ABB RobotStudio station: stationlab5.rsstn

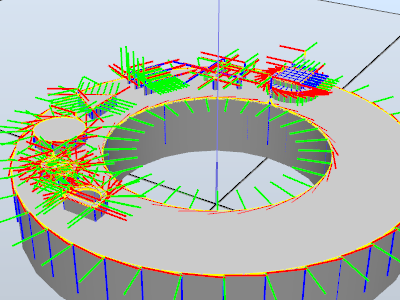
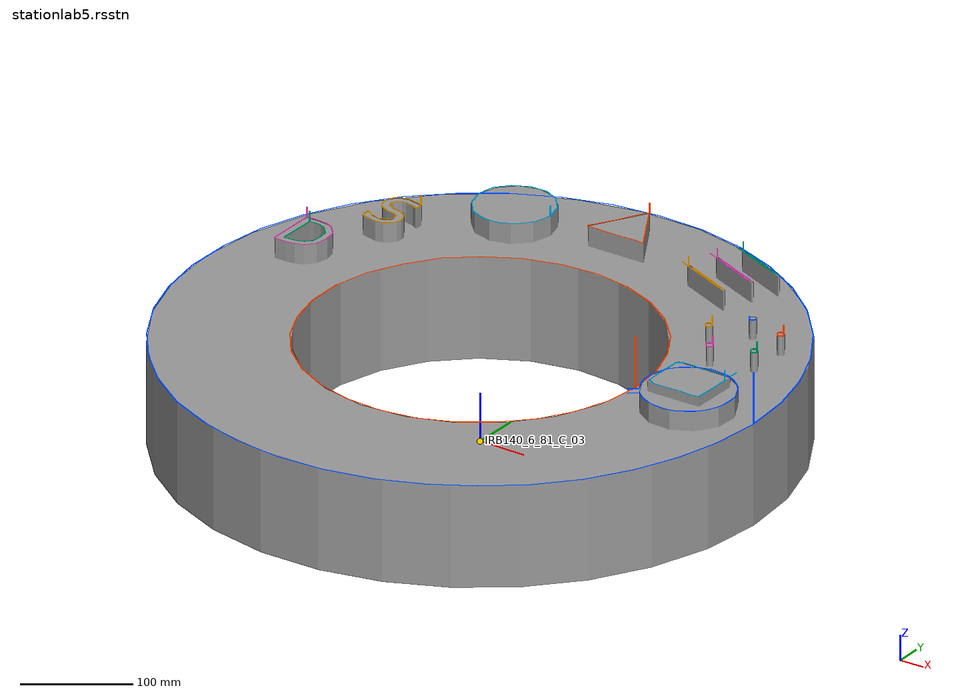
[picture v1: parts stored in the station drawn from their meshes, with robot base, taught points and paths (robot models come from the ABB library and are not in the file)]
Station Station (saved by RobotStudio 22.2.9947.0)
Controller lab5_controller
  mechanical unit ROB_1: IRB140_6_81_C_03, 6 joints, base frame (0, 0, 0) mm
Layout (positions relative to the parent item):
  - IRB140_6_81_C_03 [mechanism, from Robots\IRB140_6_81_C_G_03.rslib] at (0, 0, 0) mm; joint values [0, 0, 0, 0, 0.5236, 0] (rad or m)
  - ToolM_DS109 [mechanism, from Lab1\ToolM_DS109.rslib] at (506.29, 0, 679.5) mm, rotated rx 180 ry 60 rz 180 deg
  - lab5CADfiguras [part], size 590 x 586.8 x 130 mm
Attachment: ToolM_DS109 is attached to IRB140_6_81_C_03 / Link6
Attachment: Workobject_2 is attached to lab5CADfiguras
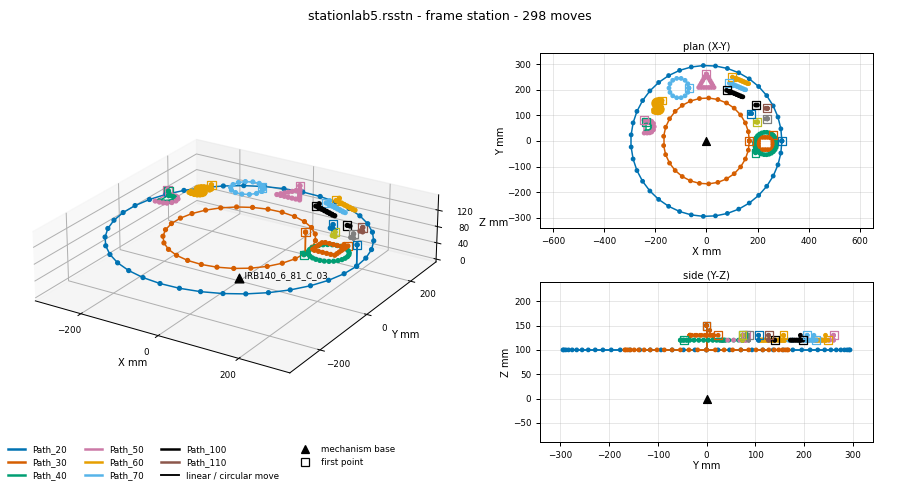
[picture p0: tool path of stationlab5.rsstn in frame station, 298 of 298 moves have a stored position in this frame; points joined in program order, loops and branches not executed]
Targets, tools, work objects and paths stored in the station, written as RAPID:
! task T_ROB1
MODULE CalibData
  PERS tooldata ToolM_DS109:=[TRUE,[[0,0,199.132],[0.949782708,0.067451832,-0.305553692,-0.000003594]],[0.13,[-0.003,72.016,0.062],[1,0,0,0],0,0,0]];
  TASK PERS wobjdata Workobject_1:=[FALSE,TRUE,"",[[0,0,0],[1,0,0,0]],[[0,0,0],[1,0,0,0]]];
  TASK PERS wobjdata Workobject_2:=[FALSE,TRUE,"",[[0,0,0],[1,0,0,0]],[[0,0,0],[1,0,0,0]]];
ENDMODULE

! task T_ROB1
MODULE Module1
  CONST robtarget Target_80_outter_ring_starts:=[[295,0,150],[0,0.707106781,0.707106781,0],[0,0,0,0],[9E+09,9E+09,9E+09,9E+09,9E+09,9E+09]];
  CONST robtarget Target_90:=[[295,0,100],[0,0.707106781,0.707106781,0],[0,0,0,0],[9E+09,9E+09,9E+09,9E+09,9E+09,9E+09]];
  CONST robtarget Target_100:=[[291.179827478,47.321327853,100],[0,0.647915395,0.761712308,0],[0,0,0,0],[9E+09,9E+09,9E+09,9E+09,9E+09,9E+09]];
  CONST robtarget Target_110:=[[279.818250374,93.417058171,100],[0,0.58452203,0.811377839,0],[0,0,0,0],[9E+09,9E+09,9E+09,9E+09,9E+09,9E+09]];
  CONST robtarget Target_120:=[[261.209527568,137.093335753,100],[0,0.517337814,0.855781272,0],[0,0,0,0],[9E+09,9E+09,9E+09,9E+09,9E+09,9E+09]];
  CONST robtarget Target_130:=[[235.835615204,177.21896795,100],[0,0.446798465,0.894634636,0],[0,0,0,0],[9E+09,9E+09,9E+09,9E+09,9E+09,9E+09]];
  CONST robtarget Target_140:=[[204.353684285,212.754721966,100],[0,0.373361455,0.927685951,0],[0,0,0,0],[9E+09,9E+09,9E+09,9E+09,9E+09,9E+09]];
  CONST robtarget Target_150:=[[167.579100286,242.780240439,100],[0,0.297503054,0.954720867,0],[0,0,0,0],[9E+09,9E+09,9E+09,9E+09,9E+09,9E+09]];
  CONST robtarget Target_160:=[[126.464305614,266.51787821,100],[0,0.219715231,0.975564051,0],[0,0,0,0],[9E+09,9E+09,9E+09,9E+09,9E+09,9E+09]];
  CONST robtarget Target_170:=[[82.074151855,283.352842931,100],[0,0.14050247,0.990080328,0],[0,0,0,0],[9E+09,9E+09,9E+09,9E+09,9E+09,9E+09]];
  CONST robtarget Target_180:=[[35.558320675,292.849117859,100],[0,0.060378497,0.998175554,0],[0,0,0,0],[9E+09,9E+09,9E+09,9E+09,9E+09,9E+09]];
  CONST robtarget Target_190:=[[-11.878452332,294.760754461,100],[0,-0.020137053,0.999797229,0],[0,0,0,0],[9E+09,9E+09,9E+09,9E+09,9E+09,9E+09]];
  CONST robtarget Target_200:=[[-59.007579664,289.038242352,100],[0,-0.100522007,0.994934835,0],[0,0,0,0],[9E+09,9E+09,9E+09,9E+09,9E+09,9E+09]];
  CONST robtarget Target_210:=[[-104.608441678,275.829791592,100],[0,-0.180255038,0.983619907,0],[0,0,0,0],[9E+09,9E+09,9E+09,9E+09,9E+09,9E+09]];
  CONST robtarget Target_220:=[[-147.5,255.477494116,100],[0,-0.258819045,0.965925826,0],[0,0,0,0],[9E+09,9E+09,9E+09,9E+09,9E+09,9E+09]];
  CONST robtarget Target_230:=[[-186.571385801,228.508463739,100],[0,-0.335704512,0.941967346,0],[0,0,0,0],[9E+09,9E+09,9E+09,9E+09,9E+09,9E+09]];
  CONST robtarget Target_240:=[[-220.81067071,195.621184181,100],[0,-0.410412805,0.911899846,0],[0,0,0,0],[9E+09,9E+09,9E+09,9E+09,9E+09,9E+09]];
  CONST robtarget Target_250:=[[-249.331075235,157.667418708,100],[0,-0.482459415,0.875918326,0],[0,0,0,0],[9E+09,9E+09,9E+09,9E+09,9E+09,9E+09]];
  CONST robtarget Target_260:=[[-271.393935879,115.630149909,100],[0,-0.55137709,0.834256139,0],[0,0,0,0],[9E+09,9E+09,9E+09,9E+09,9E+09,9E+09]];
  CONST robtarget Target_270:=[[-286.427836141,70.598120965,100],[0,-0.616718873,0.787183481,0],[0,0,0,0],[9E+09,9E+09,9E+09,9E+09,9E+09,9E+09]];
  CONST robtarget Target_280_outter_ring_half:=[[-294.0434059,23.737637771,100],[0,-0.678060997,0.735005636,0],[0,0,0,0],[9E+09,9E+09,9E+09,9E+09,9E+09,9E+09]];
  CONST robtarget Target_290:=[[-294.0434059,-23.737637771,100],[0,0.735005636,-0.678060997,0],[0,0,0,0],[9E+09,9E+09,9E+09,9E+09,9E+09,9E+09]];
  CONST robtarget Target_300:=[[-286.427836141,-70.598120965,100],[0,0.787183481,-0.616718873,0],[0,0,0,0],[9E+09,9E+09,9E+09,9E+09,9E+09,9E+09]];
  CONST robtarget Target_310:=[[-271.393935879,-115.630149909,100],[0,0.834256139,-0.55137709,0],[0,0,0,0],[9E+09,9E+09,9E+09,9E+09,9E+09,9E+09]];
  CONST robtarget Target_320:=[[-249.331075235,-157.667418708,100],[0,0.875918326,-0.482459415,0],[0,0,0,0],[9E+09,9E+09,9E+09,9E+09,9E+09,9E+09]];
  CONST robtarget Target_330:=[[-220.81067071,-195.621184181,100],[0,0.911899846,-0.410412805,0],[0,0,0,0],[9E+09,9E+09,9E+09,9E+09,9E+09,9E+09]];
  CONST robtarget Target_340:=[[-186.571385801,-228.508463739,100],[0,0.941967346,-0.335704512,0],[0,0,0,0],[9E+09,9E+09,9E+09,9E+09,9E+09,9E+09]];
  CONST robtarget Target_350:=[[-147.5,-255.477494116,100],[0,0.965925826,-0.258819045,0],[0,0,0,0],[9E+09,9E+09,9E+09,9E+09,9E+09,9E+09]];
  CONST robtarget Target_360:=[[-104.608441678,-275.829791592,100],[0,0.983619907,-0.180255038,0],[0,0,0,0],[9E+09,9E+09,9E+09,9E+09,9E+09,9E+09]];
  CONST robtarget Target_370:=[[-59.007579664,-289.038242352,100],[0,0.994934835,-0.100522007,0],[0,0,0,0],[9E+09,9E+09,9E+09,9E+09,9E+09,9E+09]];
  CONST robtarget Target_380:=[[-11.878452332,-294.760754461,100],[0,0.999797229,-0.020137053,0],[0,0,0,0],[9E+09,9E+09,9E+09,9E+09,9E+09,9E+09]];
  CONST robtarget Target_390:=[[35.558320675,-292.849117859,100],[0,0.998175554,0.060378497,0],[0,0,0,0],[9E+09,9E+09,9E+09,9E+09,9E+09,9E+09]];
  CONST robtarget Target_400:=[[82.074151855,-283.352842931,100],[0,0.990080328,0.14050247,0],[0,0,0,0],[9E+09,9E+09,9E+09,9E+09,9E+09,9E+09]];
  CONST robtarget Target_410:=[[126.464305614,-266.51787821,100],[0,0.975564051,0.219715231,0],[0,0,0,0],[9E+09,9E+09,9E+09,9E+09,9E+09,9E+09]];
  CONST robtarget Target_420:=[[167.579100286,-242.780240439,100],[0,0.954720867,0.297503054,0],[0,0,0,0],[9E+09,9E+09,9E+09,9E+09,9E+09,9E+09]];
  CONST robtarget Target_430:=[[204.353684285,-212.754721966,100],[0,0.927685951,0.373361455,0],[0,0,0,0],[9E+09,9E+09,9E+09,9E+09,9E+09,9E+09]];
  CONST robtarget Target_440:=[[235.835615204,-177.21896795,100],[0,0.894634636,0.446798465,0],[0,0,0,0],[9E+09,9E+09,9E+09,9E+09,9E+09,9E+09]];
  CONST robtarget Target_450:=[[261.209527568,-137.093335753,100],[0,0.855781272,0.517337814,0],[0,0,0,0],[9E+09,9E+09,9E+09,9E+09,9E+09,9E+09]];
  CONST robtarget Target_460:=[[279.818250374,-93.417058171,100],[0,0.811377839,0.58452203,0],[0,0,0,0],[9E+09,9E+09,9E+09,9E+09,9E+09,9E+09]];
  CONST robtarget Target_470:=[[291.179827478,-47.321327853,100],[0,0.761712308,0.647915395,0],[0,0,0,0],[9E+09,9E+09,9E+09,9E+09,9E+09,9E+09]];
  CONST robtarget Target_480:=[[295,0,100],[0,0.707106781,0.707106781,0],[0,0,0,0],[9E+09,9E+09,9E+09,9E+09,9E+09,9E+09]];
  CONST robtarget Target_490_outer_ring_ends:=[[295,0,150],[0,0.707106781,0.707106781,0],[0,0,0,0],[9E+09,9E+09,9E+09,9E+09,9E+09,9E+09]];
  CONST robtarget Target_500_inner_ring_starts:=[[168,0,150],[0,-0.707106781,0.707106781,0],[0,0,0,0],[9E+09,9E+09,9E+09,9E+09,9E+09,9E+09]];
  CONST robtarget Target_510:=[[168,0,100],[0,-0.707106781,0.707106781,0],[0,0,0,0],[9E+09,9E+09,9E+09,9E+09,9E+09,9E+09]];
  CONST robtarget Target_520:=[[164.072253359,-36.115033955,100],[0,-0.62651,0.779413382,0],[0,0,0,0],[9E+09,9E+09,9E+09,9E+09,9E+09,9E+09]];
  CONST robtarget Target_530:=[[152.472670505,-70.541369062,100],[0,-0.538567962,0.842582074,0],[0,0,0,0],[9E+09,9E+09,9E+09,9E+09,9E+09,9E+09]];
  CONST robtarget Target_540:=[[133.743635039,-101.669268153,100],[0,-0.444311706,0.895872261,0],[0,0,0,0],[9E+09,9E+09,9E+09,9E+09,9E+09,9E+09]];
  CONST robtarget Target_550:=[[108.760895843,-128.043225261,100],[0,-0.344846303,0.938659165,0],[0,0,0,0],[9E+09,9E+09,9E+09,9E+09,9E+09,9E+09]];
  CONST robtarget Target_560:=[[78.692618038,-148.430023467,100],[0,-0.241337891,0.970441148,0],[0,0,0,0],[9E+09,9E+09,9E+09,9E+09,9E+09,9E+09]];
  CONST robtarget Target_570:=[[44.944760873,-161.876398743,100],[0,-0.135000014,0.990845597,0],[0,0,0,0],[9E+09,9E+09,9E+09,9E+09,9E+09,9E+09]];
  CONST robtarget Target_580:=[[9.095336642,-167.753613527,100],[0,-0.027079385,0.999633286,0],[0,0,0,0],[9E+09,9E+09,9E+09,9E+09,9E+09,9E+09]];
  CONST robtarget Target_590:=[[-27.179375421,-165.786855787,100],[0,0.081158726,0.99670119,0],[0,0,0,0],[9E+09,9E+09,9E+09,9E+09,9E+09,9E+09]];
  CONST robtarget Target_600:=[[-62.183210097,-156.068088929,100],[0,0.188445324,0.982083683,0],[0,0,0,0],[9E+09,9E+09,9E+09,9E+09,9E+09,9E+09]];
  CONST robtarget Target_610:=[[-94.279426981,-139.05175169,100],[0,0.293522573,0.955952143,0],[0,0,0,0],[9E+09,9E+09,9E+09,9E+09,9E+09,9E+09]];
  CONST robtarget Target_620:=[[-121.967242643,-115.533509087,100],[0,0.395158539,0.918612938,0],[0,0,0,0],[9E+09,9E+09,9E+09,9E+09,9E+09,9E+09]];
  CONST robtarget Target_630:=[[-143.952005596,-86.613048006,100],[0,0.492161631,0.870503836,0],[0,0,0,0],[9E+09,9E+09,9E+09,9E+09,9E+09,9E+09]];
  CONST robtarget Target_640:=[[-159.205732759,-53.642657063,100],[0,0.583394579,0.812188873,0],[0,0,0,0],[9E+09,9E+09,9E+09,9E+09,9E+09,9E+09]];
  CONST robtarget Target_650_inner_ring_half:=[[-167.015176802,-18.163995095,100],[0,0.667787759,0.744351738,0],[0,0,0,0],[9E+09,9E+09,9E+09,9E+09,9E+09,9E+09]];
  CONST robtarget Target_660:=[[-167.015176802,18.163995095,100],[0,0.744351738,0.667787759,0],[0,0,0,0],[9E+09,9E+09,9E+09,9E+09,9E+09,9E+09]];
  CONST robtarget Target_670:=[[-159.205732759,53.642657063,100],[0,0.812188873,0.583394579,0],[0,0,0,0],[9E+09,9E+09,9E+09,9E+09,9E+09,9E+09]];
  CONST robtarget Target_680:=[[-143.952005596,86.613048006,100],[0,0.870503836,0.492161631,0],[0,0,0,0],[9E+09,9E+09,9E+09,9E+09,9E+09,9E+09]];
  CONST robtarget Target_690:=[[-121.967242643,115.533509087,100],[0,0.918612938,0.395158539,0],[0,0,0,0],[9E+09,9E+09,9E+09,9E+09,9E+09,9E+09]];
  CONST robtarget Target_700:=[[-94.279426981,139.05175169,100],[0,0.955952143,0.293522573,0],[0,0,0,0],[9E+09,9E+09,9E+09,9E+09,9E+09,9E+09]];
  CONST robtarget Target_710:=[[-62.183210097,156.068088929,100],[0,0.982083683,0.188445324,0],[0,0,0,0],[9E+09,9E+09,9E+09,9E+09,9E+09,9E+09]];
  CONST robtarget Target_720:=[[-27.179375421,165.786855787,100],[0,0.99670119,0.081158726,0],[0,0,0,0],[9E+09,9E+09,9E+09,9E+09,9E+09,9E+09]];
  CONST robtarget Target_730:=[[9.095336642,167.753613527,100],[0,0.999633286,-0.027079385,0],[0,0,0,0],[9E+09,9E+09,9E+09,9E+09,9E+09,9E+09]];
  CONST robtarget Target_740:=[[44.944760873,161.876398743,100],[0,0.990845597,-0.135000014,0],[0,0,0,0],[9E+09,9E+09,9E+09,9E+09,9E+09,9E+09]];
  CONST robtarget Target_750:=[[78.692618038,148.430023467,100],[0,0.970441148,-0.241337891,0],[0,0,0,0],[9E+09,9E+09,9E+09,9E+09,9E+09,9E+09]];
  CONST robtarget Target_760:=[[108.760895843,128.043225261,100],[0,0.938659165,-0.344846303,0],[0,0,0,0],[9E+09,9E+09,9E+09,9E+09,9E+09,9E+09]];
  CONST robtarget Target_770:=[[133.743635039,101.669268153,100],[0,0.895872261,-0.444311706,0],[0,0,0,0],[9E+09,9E+09,9E+09,9E+09,9E+09,9E+09]];
  CONST robtarget Target_780:=[[152.472670505,70.541369062,100],[0,0.842582074,-0.538567962,0],[0,0,0,0],[9E+09,9E+09,9E+09,9E+09,9E+09,9E+09]];
  CONST robtarget Target_790:=[[164.072253359,36.115033955,100],[0,0.779413382,-0.62651,0],[0,0,0,0],[9E+09,9E+09,9E+09,9E+09,9E+09,9E+09]];
  CONST robtarget Target_800:=[[168,0,100],[0,-0.707106781,0.707106781,0],[0,0,0,0],[9E+09,9E+09,9E+09,9E+09,9E+09,9E+09]];
  CONST robtarget Target_810_inner_ring_ends:=[[168,0,150],[0,-0.707106781,0.707106781,0],[0,0,0,0],[9E+09,9E+09,9E+09,9E+09,9E+09,9E+09]];
  CONST robtarget Target_810:=[[-236.504880452,74.974751988,130],[0,-0.707106781,0.707106781,0],[0,0,0,0],[9E+09,9E+09,9E+09,9E+09,9E+09,9E+09]];
  CONST robtarget Target_820_d_inner_starts:=[[-236.504880452,74.974751988,120],[0,-0.707106781,0.707106781,0],[0,0,0,0],[9E+09,9E+09,9E+09,9E+09,9E+09,9E+09]];
  CONST robtarget Target_830:=[[-236.504880452,36.482045343,120],[0,-0.707106781,0.707106781,0],[0,0,0,0],[9E+09,9E+09,9E+09,9E+09,9E+09,9E+09]];
  CONST robtarget Target_840:=[[-231.440050631,36.482045343,120],[0,1,0,0],[0,0,0,0],[9E+09,9E+09,9E+09,9E+09,9E+09,9E+09]];
  CONST robtarget Target_850:=[[-223.680731344,37.191121518,120],[0,0.994543645,0.104321318,0],[0,0,0,0],[9E+09,9E+09,9E+09,9E+09,9E+09,9E+09]];
  CONST robtarget Target_860:=[[-217.623194877,39.804573706,120],[0,0.953587299,0.301116693,0],[0,0,0,0],[9E+09,9E+09,9E+09,9E+09,9E+09,9E+09]];
  CONST robtarget Target_870:=[[-212.396290501,46.044444047,120],[0,0.839280324,0.54369894,0],[0,0,0,0],[9E+09,9E+09,9E+09,9E+09,9E+09,9E+09]];
  CONST robtarget Target_880:=[[-210.653989042,55.768917304,120],[0,0.707106781,0.707106781,0],[0,0,0,0],[9E+09,9E+09,9E+09,9E+09,9E+09,9E+09]];
  CONST robtarget Target_890:=[[-212.558365055,65.594687159,120],[0,0.536830761,0.843689951,0],[0,0,0,0],[9E+09,9E+09,9E+09,9E+09,9E+09,9E+09]];
  CONST robtarget Target_900:=[[-218.230974456,71.976372734,120],[0,0.271476286,0.962445129,0],[0,0,0,0],[9E+09,9E+09,9E+09,9E+09,9E+09,9E+09]];
  CONST robtarget Target_910:=[[-223.923843175,74.265675813,120],[0,0.115102592,0.993353609,0],[0,0,0,0],[9E+09,9E+09,9E+09,9E+09,9E+09,9E+09]];
  CONST robtarget Target_920:=[[-231.440050631,74.974751988,120],[0,0,1,0],[0,0,0,0],[9E+09,9E+09,9E+09,9E+09,9E+09,9E+09]];
  CONST robtarget Target_930:=[[-236.504880452,74.974751988,120],[0,0,1,0],[0,0,0,0],[9E+09,9E+09,9E+09,9E+09,9E+09,9E+09]];
  CONST robtarget Target_940_d_inner:=[[-236.504880452,74.974751988,130],[0,0,1,0],[0,0,0,0],[9E+09,9E+09,9E+09,9E+09,9E+09,9E+09]];
  CONST robtarget Target_940:=[[-243.149937179,80.728398666,130],[0,-0.707106781,0.707106781,0],[0,0,0,0],[9E+09,9E+09,9E+09,9E+09,9E+09,9E+09]];
  CONST robtarget Target_950_d_outter_starts:=[[-243.149937179,80.728398666,120],[0,-0.707106781,0.707106781,0],[0,0,0,0],[9E+09,9E+09,9E+09,9E+09,9E+09,9E+09]];
  CONST robtarget Target_960:=[[-243.149937179,30.728398666,120],[0,-0.707106781,0.707106781,0],[0,0,0,0],[9E+09,9E+09,9E+09,9E+09,9E+09,9E+09]];
  CONST robtarget Target_970:=[[-231.642643824,30.728398666,120],[0,1,0,0],[0,0,0,0],[9E+09,9E+09,9E+09,9E+09,9E+09,9E+09]];
  CONST robtarget Target_980:=[[-221.654799415,31.538771437,120],[0,0.994784133,0.102002596,0],[0,0,0,0],[9E+09,9E+09,9E+09,9E+09,9E+09,9E+09]];
  CONST robtarget Target_990:=[[-213.935998767,34.739743885,120],[0,0.960985001,0.276600484,0],[0,0,0,0],[9E+09,9E+09,9E+09,9E+09,9E+09,9E+09]];
  CONST robtarget Target_1000:=[[-206.500828589,43.329695262,120],[0,0.851421887,0.524481429,0],[0,0,0,0],[9E+09,9E+09,9E+09,9E+09,9E+09,9E+09]];
  CONST robtarget Target_1010:=[[-203.725301846,55.687880027,120],[0,0.707106781,0.707106781,0],[0,0,0,0],[9E+09,9E+09,9E+09,9E+09,9E+09,9E+09]];
  CONST robtarget Target_1020:=[[-206.379272673,68.268917304,120],[0,0.525079618,0.851053109,0],[0,0,0,0],[9E+09,9E+09,9E+09,9E+09,9E+09,9E+09]];
  CONST robtarget Target_1030:=[[-213.85496149,76.757572086,120],[0,0.288854798,0.957372919,0],[0,0,0,0],[9E+09,9E+09,9E+09,9E+09,9E+09,9E+09]];
  CONST robtarget Target_1040:=[[-220.702611409,79.674914063,120],[0,0.128060594,0.991766346,0],[0,0,0,0],[9E+09,9E+09,9E+09,9E+09,9E+09,9E+09]];
  CONST robtarget Target_1050:=[[-231.764199739,80.728398666,120],[0,0,1,0],[0,0,0,0],[9E+09,9E+09,9E+09,9E+09,9E+09,9E+09]];
  CONST robtarget Target_1060:=[[-243.149937179,80.728398666,120],[0,0,1,0],[0,0,0,0],[9E+09,9E+09,9E+09,9E+09,9E+09,9E+09]];
  CONST robtarget Target_1070_d_outter_ends:=[[-243.149937179,80.728398666,130],[0,0,1,0],[0,0,0,0],[9E+09,9E+09,9E+09,9E+09,9E+09,9E+09]];
  CONST robtarget Target_1070:=[[-174.142803292,158.219300938,130],[0,0.227282029,0.973828978,0],[0,0,0,0],[9E+09,9E+09,9E+09,9E+09,9E+09,9E+09]];
  CONST robtarget Target_1080_s_starts:=[[-174.142803292,158.219300938,120],[0,0.227282029,0.973828978,0],[0,0,0,0],[9E+09,9E+09,9E+09,9E+09,9E+09,9E+09]];
  CONST robtarget Target_1090:=[[-181.071490488,160.630159933,120],[0,0.109402737,0.993997506,0],[0,0,0,0],[9E+09,9E+09,9E+09,9E+09,9E+09,9E+09]];
  CONST robtarget Target_1100:=[[-189.013143649,161.460792024,120],[0,0,1,0],[0,0,0,0],[9E+09,9E+09,9E+09,9E+09,9E+09,9E+09]];
  CONST robtarget Target_1110:=[[-195.698719013,160.43263157,120],[0,-0.163403874,0.98655926,0],[0,0,0,0],[9E+09,9E+09,9E+09,9E+09,9E+09,9E+09]];
  CONST robtarget Target_1120:=[[-201.087697944,157.348150208,120],[0,-0.349735999,0.936848297,0],[0,0,0,0],[9E+09,9E+09,9E+09,9E+09,9E+09,9E+09]];
  CONST robtarget Target_1130:=[[-204.643208478,152.7442199,120],[0,-0.537680352,0.843148764,0],[0,0,0,0],[9E+09,9E+09,9E+09,9E+09,9E+09,9E+09]];
  CONST robtarget Target_1140:=[[-205.828378657,147.157712607,120],[0,-0.707106781,0.707106781,0],[0,0,0,0],[9E+09,9E+09,9E+09,9E+09,9E+09,9E+09]];
  CONST robtarget Target_1150:=[[-204.977487247,142.011845508,120],[0,0.823620533,-0.567141267,0],[0,0,0,0],[9E+09,9E+09,9E+09,9E+09,9E+09,9E+09]];
  CONST robtarget Target_1160:=[[-202.586887571,138.122056205,120],[0,0.916450944,-0.400147057,0],[0,0,0,0],[9E+09,9E+09,9E+09,9E+09,9E+09,9E+09]];
  CONST robtarget Target_1170:=[[-198.960469418,135.42756674,120],[0,0.972793034,-0.231675878,0],[0,0,0,0],[9E+09,9E+09,9E+09,9E+09,9E+09,9E+09]];
  CONST robtarget Target_1180:=[[-194.321085302,133.705524601,120],[0,0.991585883,-0.129450518,0],[0,0,0,0],[9E+09,9E+09,9E+09,9E+09,9E+09,9E+09]];
  CONST robtarget Target_1190:=[[-185.2854289,131.43648084,120],[0,0.990653418,-0.136403098,0],[0,0,0,0],[9E+09,9E+09,9E+09,9E+09,9E+09,9E+09]];
  CONST robtarget Target_1200:=[[-180.605526145,128.640694779,120],[0,0.900437375,-0.43498567,0],[0,0,0,0],[9E+09,9E+09,9E+09,9E+09,9E+09,9E+09]];
  CONST robtarget Target_1210:=[[-179.126595837,123.77845815,120],[0,-0.707106781,0.707106781,0],[0,0,0,0],[9E+09,9E+09,9E+09,9E+09,9E+09,9E+09]];
  CONST robtarget Target_1220:=[[-181.942641218,117.720921683,120],[0,-0.334706425,0.942322455,0],[0,0,0,0],[9E+09,9E+09,9E+09,9E+09,9E+09,9E+09]];
  CONST robtarget Target_1230:=[[-190.269221444,115.431618604,120],[0,0,1,0],[0,0,0,0],[9E+09,9E+09,9E+09,9E+09,9E+09,9E+09]];
  CONST robtarget Target_1240:=[[-198.271652563,117.133401424,120],[0,0.193221244,0.981155212,0],[0,0,0,0],[9E+09,9E+09,9E+09,9E+09,9E+09,9E+09]];
  CONST robtarget Target_1250:=[[-205.706822741,121.914600776,120],[0,0.367929084,0.929853854,0],[0,0,0,0],[9E+09,9E+09,9E+09,9E+09,9E+09,9E+09]];
  CONST robtarget Target_1260:=[[-206.193046404,121.914600776,120],[0,0,1,0],[0,0,0,0],[9E+09,9E+09,9E+09,9E+09,9E+09,9E+09]];
  CONST robtarget Target_1270:=[[-206.193046404,113.567761229,120],[0,-0.707106781,0.707106781,0],[0,0,0,0],[9E+09,9E+09,9E+09,9E+09,9E+09,9E+09]];
  CONST robtarget Target_1280:=[[-199.021247376,110.812493806,120],[0,0.989541733,-0.144246866,0],[0,0,0,0],[9E+09,9E+09,9E+09,9E+09,9E+09,9E+09]];
  CONST robtarget Target_1290:=[[-189.782997782,109.677971926,120],[0,1,0,0],[0,0,0,0],[9E+09,9E+09,9E+09,9E+09,9E+09,9E+09]];
  CONST robtarget Target_1300:=[[-182.16549373,110.853012445,120],[0,0.983031812,0.183435159,0],[0,0,0,0],[9E+09,9E+09,9E+09,9E+09,9E+09,9E+09]];
  CONST robtarget Target_1310:=[[-176.735996161,114.216059447,120],[0,0.932113972,0.362165078,0],[0,0,0,0],[9E+09,9E+09,9E+09,9E+09,9E+09,9E+09]];
  CONST robtarget Target_1320:=[[-173.393208478,119.037777437,120],[0,0.833172024,0.553013904,0],[0,0,0,0],[9E+09,9E+09,9E+09,9E+09,9E+09,9E+09]];
  CONST robtarget Target_1330:=[[-172.197908641,124.831942753,120],[0,0.707106781,0.707106781,0],[0,0,0,0],[9E+09,9E+09,9E+09,9E+09,9E+09,9E+09]];
  CONST robtarget Target_1340:=[[-174.588508316,132.672299317,120],[0,0.446758127,0.89465478,0],[0,0,0,0],[9E+09,9E+09,9E+09,9E+09,9E+09,9E+09]];
  CONST robtarget Target_1350:=[[-182.124975091,137.433239349,120],[0,0.148422353,0.988924064,0],[0,0,0,0],[9E+09,9E+09,9E+09,9E+09,9E+09,9E+09]];
  CONST robtarget Target_1360:=[[-192.37619065,140.066950857,120],[0,0.131118728,0.991366672,0],[0,0,0,0],[9E+09,9E+09,9E+09,9E+09,9E+09,9E+09]];
  CONST robtarget Target_1370:=[[-197.21816796,142.80195896,120],[0,0.408744216,0.912648983,0],[0,0,0,0],[9E+09,9E+09,9E+09,9E+09,9E+09,9E+09]];
  CONST robtarget Target_1380:=[[-198.899691461,147.846529463,120],[0,0.707106781,0.707106781,0],[0,0,0,0],[9E+09,9E+09,9E+09,9E+09,9E+09,9E+09]];
  CONST robtarget Target_1390:=[[-196.043127441,153.539398182,120],[0,0.947786225,0.318906369,0],[0,0,0,0],[9E+09,9E+09,9E+09,9E+09,9E+09,9E+09]];
  CONST robtarget Target_1400:=[[-188.567438624,155.707145346,120],[0,1,0,0],[0,0,0,0],[9E+09,9E+09,9E+09,9E+09,9E+09,9E+09]];
  CONST robtarget Target_1410:=[[-180.74734138,154.086399803,120],[0,0.979048021,-0.203629497,0],[0,0,0,0],[9E+09,9E+09,9E+09,9E+09,9E+09,9E+09]];
  CONST robtarget Target_1420:=[[-174.142803292,150.277647777,120],[0,1,0,0],[0,0,0,0],[9E+09,9E+09,9E+09,9E+09,9E+09,9E+09]];
  CONST robtarget Target_1430:=[[-174.142803292,158.219300938,120],[0,0.707106781,0.707106781,0],[0,0,0,0],[9E+09,9E+09,9E+09,9E+09,9E+09,9E+09]];
  CONST robtarget Target_1440_s_ends:=[[-174.142803292,158.219300938,130],[0,0.707106781,0.707106781,0],[0,0,0,0],[9E+09,9E+09,9E+09,9E+09,9E+09,9E+09]];
  CONST robtarget Target_1440:=[[-68.753776769,206.725037499,130],[0,0.707106781,0.707106781,0],[0,0,0,0],[9E+09,9E+09,9E+09,9E+09,9E+09,9E+09]];
  CONST robtarget Target_1450_circle_starts:=[[-68.753776769,206.725037499,120],[0,0.707106781,0.707106781,0],[0,0,0,0],[9E+09,9E+09,9E+09,9E+09,9E+09,9E+09]];
  CONST robtarget Target_1460:=[[-72.586344164,223.516612395,120],[0,0.532032077,0.846724199,0],[0,0,0,0],[9E+09,9E+09,9E+09,9E+09,9E+09,9E+09]];
  CONST robtarget Target_1470:=[[-83.324959372,236.982409948,120],[0,0.330279062,0.94388333,0],[0,0,0,0],[9E+09,9E+09,9E+09,9E+09,9E+09,9E+09]];
  CONST robtarget Target_1480:=[[-98.842707952,244.455363805,120],[0,0.111964476,0.99371221,0],[0,0,0,0],[9E+09,9E+09,9E+09,9E+09,9E+09,9E+09]];
  CONST robtarget Target_1490:=[[-116.066109483,244.455363805,120],[0,-0.111964476,0.99371221,0],[0,0,0,0],[9E+09,9E+09,9E+09,9E+09,9E+09,9E+09]];
  CONST robtarget Target_1500:=[[-131.583858063,236.982409948,120],[0,-0.330279062,0.94388333,0],[0,0,0,0],[9E+09,9E+09,9E+09,9E+09,9E+09,9E+09]];
  CONST robtarget Target_1510:=[[-142.322473271,223.516612395,120],[0,-0.532032077,0.846724199,0],[0,0,0,0],[9E+09,9E+09,9E+09,9E+09,9E+09,9E+09]];
  CONST robtarget Target_1520:=[[-146.155040666,206.725037499,120],[0,-0.707106781,0.707106781,0],[0,0,0,0],[9E+09,9E+09,9E+09,9E+09,9E+09,9E+09]];
  CONST robtarget Target_1530:=[[-142.322473271,189.933462603,120],[0,0.846724199,-0.532032077,0],[0,0,0,0],[9E+09,9E+09,9E+09,9E+09,9E+09,9E+09]];
  CONST robtarget Target_1540:=[[-131.583858063,176.46766505,120],[0,0.94388333,-0.330279062,0],[0,0,0,0],[9E+09,9E+09,9E+09,9E+09,9E+09,9E+09]];
  CONST robtarget Target_1550:=[[-116.066109483,168.994711193,120],[0,0.99371221,-0.111964476,0],[0,0,0,0],[9E+09,9E+09,9E+09,9E+09,9E+09,9E+09]];
  CONST robtarget Target_1560:=[[-98.842707952,168.994711193,120],[0,0.99371221,0.111964476,0],[0,0,0,0],[9E+09,9E+09,9E+09,9E+09,9E+09,9E+09]];
  CONST robtarget Target_1570:=[[-83.324959372,176.46766505,120],[0,0.94388333,0.330279062,0],[0,0,0,0],[9E+09,9E+09,9E+09,9E+09,9E+09,9E+09]];
  CONST robtarget Target_1580:=[[-72.586344164,189.933462603,120],[0,0.846724199,0.532032077,0],[0,0,0,0],[9E+09,9E+09,9E+09,9E+09,9E+09,9E+09]];
  CONST robtarget Target_1590:=[[-68.753776769,206.725037499,120],[0,0.707106781,0.707106781,0],[0,0,0,0],[9E+09,9E+09,9E+09,9E+09,9E+09,9E+09]];
  CONST robtarget Target_1600_circle_ends:=[[-68.753776769,206.725037499,130],[0,0.707106781,0.707106781,0],[0,0,0,0],[9E+09,9E+09,9E+09,9E+09,9E+09,9E+09]];
  CONST robtarget Target_2450_point1_starts:=[[195.937959768,143.518538082,120],[0,0,-0.707106781,0.707106781],[0,0,0,0],[9E+09,9E+09,9E+09,9E+09,9E+09,9E+09]];
  CONST robtarget Target_2460:=[[192.506872882,140.087451197,120],[0.5,-0.5,0.5,-0.5],[0,0,0,0],[9E+09,9E+09,9E+09,9E+09,9E+09,9E+09]];
  CONST robtarget Target_2470:=[[195.937959768,136.656364312,120],[0.707106781,-0.707106781,0,0],[0,0,0,0],[9E+09,9E+09,9E+09,9E+09,9E+09,9E+09]];
  CONST robtarget Target_2480_point1_ends:=[[199.369046653,140.087451197,120],[0.5,-0.5,-0.5,0.5],[0,0,0,0],[9E+09,9E+09,9E+09,9E+09,9E+09,9E+09]];
  CONST robtarget Target_2480:=[[238.2927152,127.440384636,130],[0,0.707106781,0.707106781,0],[0,0,0,0],[9E+09,9E+09,9E+09,9E+09,9E+09,9E+09]];
  CONST robtarget Target_2490_point2_starts:=[[238.2927152,127.440384636,120],[0,0.707106781,0.707106781,0],[0,0,0,0],[9E+09,9E+09,9E+09,9E+09,9E+09,9E+09]];
  CONST robtarget Target_2500:=[[234.861628315,130.871471522,120],[0,0,1,0],[0,0,0,0],[9E+09,9E+09,9E+09,9E+09,9E+09,9E+09]];
  CONST robtarget Target_2510:=[[231.430541429,127.440384636,120],[0,-0.707106781,0.707106781,0],[0,0,0,0],[9E+09,9E+09,9E+09,9E+09,9E+09,9E+09]];
  CONST robtarget Target_2520:=[[234.861628315,124.009297751,120],[0,1,0,0],[0,0,0,0],[9E+09,9E+09,9E+09,9E+09,9E+09,9E+09]];
  CONST robtarget Target_2530:=[[238.2927152,127.440384636,120],[0,0.707106781,0.707106781,0],[0,0,0,0],[9E+09,9E+09,9E+09,9E+09,9E+09,9E+09]];
  CONST robtarget Target_2540_point2_ends:=[[238.2927152,127.440384636,130],[0,0.707106781,0.707106781,0],[0,0,0,0],[9E+09,9E+09,9E+09,9E+09,9E+09,9E+09]];
  CONST robtarget Target_2540:=[[238.2927152,86.51361753,130],[0,0.707106781,0.707106781,0],[0,0,0,0],[9E+09,9E+09,9E+09,9E+09,9E+09,9E+09]];
  CONST robtarget Target_2550_point3_starts:=[[238.2927152,86.51361753,120],[0,0.707106781,0.707106781,0],[0,0,0,0],[9E+09,9E+09,9E+09,9E+09,9E+09,9E+09]];
  CONST robtarget Target_2560:=[[234.861628315,89.944704415,120],[0,0,1,0],[0,0,0,0],[9E+09,9E+09,9E+09,9E+09,9E+09,9E+09]];
  CONST robtarget Target_2570:=[[231.430541429,86.51361753,120],[0,-0.707106781,0.707106781,0],[0,0,0,0],[9E+09,9E+09,9E+09,9E+09,9E+09,9E+09]];
  CONST robtarget Target_2580:=[[234.861628315,83.082530645,120],[0,1,0,0],[0,0,0,0],[9E+09,9E+09,9E+09,9E+09,9E+09,9E+09]];
  CONST robtarget Target_2590:=[[238.2927152,86.51361753,120],[0,0.707106781,0.707106781,0],[0,0,0,0],[9E+09,9E+09,9E+09,9E+09,9E+09,9E+09]];
  CONST robtarget Target_2600_point3_ends:=[[238.2927152,86.51361753,130],[0,0.707106781,0.707106781,0],[0,0,0,0],[9E+09,9E+09,9E+09,9E+09,9E+09,9E+09]];
  CONST robtarget Target_2600:=[[199.369046653,73.86655097,130],[0,0.707106781,0.707106781,0],[0,0,0,0],[9E+09,9E+09,9E+09,9E+09,9E+09,9E+09]];
  CONST robtarget Target_2610_point4_starts:=[[199.369046653,73.86655097,120],[0,0.707106781,0.707106781,0],[0,0,0,0],[9E+09,9E+09,9E+09,9E+09,9E+09,9E+09]];
  CONST robtarget Target_2620:=[[195.937959768,77.297637855,120],[0,0,1,0],[0,0,0,0],[9E+09,9E+09,9E+09,9E+09,9E+09,9E+09]];
  CONST robtarget Target_2630:=[[192.506872882,73.86655097,120],[0,-0.707106781,0.707106781,0],[0,0,0,0],[9E+09,9E+09,9E+09,9E+09,9E+09,9E+09]];
  CONST robtarget Target_2640:=[[195.937959768,70.435464084,120],[0,1,0,0],[0,0,0,0],[9E+09,9E+09,9E+09,9E+09,9E+09,9E+09]];
  CONST robtarget Target_2650:=[[199.369046653,73.86655097,120],[0,0.707106781,0.707106781,0],[0,0,0,0],[9E+09,9E+09,9E+09,9E+09,9E+09,9E+09]];
  CONST robtarget Target_2660_point4_ends:=[[199.369046653,73.86655097,130],[0,0.707106781,0.707106781,0],[0,0,0,0],[9E+09,9E+09,9E+09,9E+09,9E+09,9E+09]];
  CONST robtarget Target_2660:=[[175.312896524,106.977001083,130],[0,0.707106781,0.707106781,0],[0,0,0,0],[9E+09,9E+09,9E+09,9E+09,9E+09,9E+09]];
  CONST robtarget Target_2670_point5_starts:=[[175.312896524,106.977001083,120],[0,0.707106781,0.707106781,0],[0,0,0,0],[9E+09,9E+09,9E+09,9E+09,9E+09,9E+09]];
  CONST robtarget Target_2680:=[[171.881809639,110.408087969,120],[0,0,1,0],[0,0,0,0],[9E+09,9E+09,9E+09,9E+09,9E+09,9E+09]];
  CONST robtarget Target_2690:=[[168.450722753,106.977001083,120],[0,-0.707106781,0.707106781,0],[0,0,0,0],[9E+09,9E+09,9E+09,9E+09,9E+09,9E+09]];
  CONST robtarget Target_2700:=[[171.881809639,103.545914198,120],[0,1,0,0],[0,0,0,0],[9E+09,9E+09,9E+09,9E+09,9E+09,9E+09]];
  CONST robtarget Target_2710:=[[175.312896524,106.977001083,120],[0,0.707106781,0.707106781,0],[0,0,0,0],[9E+09,9E+09,9E+09,9E+09,9E+09,9E+09]];
  CONST robtarget Target_2720_point5_ends:=[[175.312896524,106.977001083,130],[0,0.707106781,0.707106781,0],[0,0,0,0],[9E+09,9E+09,9E+09,9E+09,9E+09,9E+09]];
  CONST robtarget Target_2720:=[[259.580226634,23.931902619,130],[0,0,-0.707106781,0.707106781],[0,0,0,0],[9E+09,9E+09,9E+09,9E+09,9E+09,9E+09]];
  CONST robtarget Target_2730_custom_starts_p1:=[[259.580226634,13.931902619,130],[0,0,-0.707106781,0.707106781],[0,0,0,0],[9E+09,9E+09,9E+09,9E+09,9E+09,9E+09]];
  CONST robtarget Target_2740:=[[249.580226634,13.931902619,130],[0,0,-0.707106781,0.707106781],[0,0,0,0],[9E+09,9E+09,9E+09,9E+09,9E+09,9E+09]];
  CONST robtarget Target_2750:=[[239.580226634,13.931902619,130],[0,0,-0.707106781,0.707106781],[0,0,0,0],[9E+09,9E+09,9E+09,9E+09,9E+09,9E+09]];
  CONST robtarget Target_2760:=[[229.580226634,13.931902619,130],[0,0,-0.707106781,0.707106781],[0,0,0,0],[9E+09,9E+09,9E+09,9E+09,9E+09,9E+09]];
  CONST robtarget Target_2770:=[[219.580226634,13.931902619,130],[0,0,-0.707106781,0.707106781],[0,0,0,0],[9E+09,9E+09,9E+09,9E+09,9E+09,9E+09]];
  CONST robtarget Target_2780:=[[209.580226634,13.931902619,130],[0,0,-0.707106781,0.707106781],[0,0,0,0],[9E+09,9E+09,9E+09,9E+09,9E+09,9E+09]];
  CONST robtarget Target_2790:=[[203.897358753,9.6147705,130],[0.5,-0.5,0.5,-0.5],[0,0,0,0],[9E+09,9E+09,9E+09,9E+09,9E+09,9E+09]];
  CONST robtarget Target_2800:=[[203.897358753,-0.3852295,130],[0.5,-0.5,0.5,-0.5],[0,0,0,0],[9E+09,9E+09,9E+09,9E+09,9E+09,9E+09]];
  CONST robtarget Target_2810:=[[203.897358753,-10.3852295,130],[0.5,-0.5,0.5,-0.5],[0,0,0,0],[9E+09,9E+09,9E+09,9E+09,9E+09,9E+09]];
  CONST robtarget Target_2820:=[[203.897358753,-20.3852295,130],[0.5,-0.5,0.5,-0.5],[0,0,0,0],[9E+09,9E+09,9E+09,9E+09,9E+09,9E+09]];
  CONST robtarget Target_2830:=[[203.897358753,-30.3852295,130],[0.5,-0.5,0.5,-0.5],[0,0,0,0],[9E+09,9E+09,9E+09,9E+09,9E+09,9E+09]];
  CONST robtarget Target_2840:=[[210.25899265,-34.023595603,130],[0,1,0,0],[0,0,0,0],[9E+09,9E+09,9E+09,9E+09,9E+09,9E+09]];
  CONST robtarget Target_2850:=[[220.25899265,-34.023595603,130],[0,1,0,0],[0,0,0,0],[9E+09,9E+09,9E+09,9E+09,9E+09,9E+09]];
  CONST robtarget Target_2860:=[[230.25899265,-34.023595603,130],[0,1,0,0],[0,0,0,0],[9E+09,9E+09,9E+09,9E+09,9E+09,9E+09]];
  CONST robtarget Target_2870:=[[240.25899265,-34.023595603,130],[0,1,0,0],[0,0,0,0],[9E+09,9E+09,9E+09,9E+09,9E+09,9E+09]];
  CONST robtarget Target_2880:=[[250.25899265,-34.023595603,130],[0,1,0,0],[0,0,0,0],[9E+09,9E+09,9E+09,9E+09,9E+09,9E+09]];
  CONST robtarget Target_2890:=[[259.580226634,-33.344829588,130],[0,0.707106781,0.707106781,0],[0,0,0,0],[9E+09,9E+09,9E+09,9E+09,9E+09,9E+09]];
  CONST robtarget Target_2900:=[[259.580226634,-23.344829588,130],[0,0.707106781,0.707106781,0],[0,0,0,0],[9E+09,9E+09,9E+09,9E+09,9E+09,9E+09]];
  CONST robtarget Target_2910:=[[259.580226634,-13.344829588,130],[0,0.707106781,0.707106781,0],[0,0,0,0],[9E+09,9E+09,9E+09,9E+09,9E+09,9E+09]];
  CONST robtarget Target_2920:=[[259.580226634,-3.344829588,130],[0,0.707106781,0.707106781,0],[0,0,0,0],[9E+09,9E+09,9E+09,9E+09,9E+09,9E+09]];
  CONST robtarget Target_2930:=[[259.580226634,6.655170412,130],[0,0.707106781,0.707106781,0],[0,0,0,0],[9E+09,9E+09,9E+09,9E+09,9E+09,9E+09]];
  CONST robtarget Target_2940_custom_ends_p1:=[[259.580226634,6.655170412,140],[0,0.707106781,0.707106781,0],[0,0,0,0],[9E+09,9E+09,9E+09,9E+09,9E+09,9E+09]];
  CONST robtarget Target_2940:=[[191.931427786,-46.535928873,120],[0.64724891,-0.64724891,0.284725918,-0.284725918],[0,0,0,0],[9E+09,9E+09,9E+09,9E+09,9E+09,9E+09]];
  CONST robtarget Target_2950_custom_start_p1:=[[199.302969384,-39.778682801,120],[0.64724891,-0.64724891,0.284725918,-0.284725918],[0,0,0,0],[9E+09,9E+09,9E+09,9E+09,9E+09,9E+09]];
  CONST robtarget Target_2960:=[[206.836246505,-46.322386874,120],[0.675359235,-0.675359235,0.209499174,-0.209499174],[0,0,0,0],[9E+09,9E+09,9E+09,9E+09,9E+09,9E+09]];
  CONST robtarget Target_2970:=[[215.650203185,-51.000473537,120],[0.694758434,-0.694758434,0.131570204,-0.131570204],[0,0,0,0],[9E+09,9E+09,9E+09,9E+09,9E+09,9E+09]];
  CONST robtarget Target_2980:=[[225.291558298,-53.572359762,120],[0.705196287,-0.705196287,0.051944174,-0.051944174],[0,0,0,0],[9E+09,9E+09,9E+09,9E+09,9E+09,9E+09]];
  CONST robtarget Target_2990:=[[235.264479559,-53.905779471,120],[0.70653816,-0.70653816,-0.028351858,0.028351858],[0,0,0,0],[9E+09,9E+09,9E+09,9E+09,9E+09,9E+09]];
  CONST robtarget Target_3000:=[[245.056083011,-51.98358567,120],[0.698766747,-0.698766747,-0.108282193,0.108282193],[0,0,0,0],[9E+09,9E+09,9E+09,9E+09,9E+09,9E+09]];
  CONST robtarget Target_3010:=[[254.162809449,-47.90463228,120],[0.681982286,-0.681982286,-0.186815849,0.186815849],[0,0,0,0],[9E+09,9E+09,9E+09,9E+09,9E+09,9E+09]];
  CONST robtarget Target_3020:=[[262.116321286,-41.878690308,120],[0.656401272,-0.656401272,-0.26293986,0.26293986],[0,0,0,0],[9E+09,9E+09,9E+09,9E+09,9E+09,9E+09]];
  CONST robtarget Target_3030:=[[268.507588056,-34.215659821,120],[0.622353662,-0.622353662,-0.33567234,0.33567234],[0,0,0,0],[9E+09,9E+09,9E+09,9E+09,9E+09,9E+09]];
  CONST robtarget Target_3040:=[[273.007921897,-25.309632509,120],[0.580278619,-0.580278619,-0.404075147,0.404075147],[0,0,0,0],[9E+09,9E+09,9E+09,9E+09,9E+09,9E+09]];
  CONST robtarget Target_3050:=[[275.385881192,-15.618624472,120],[0.530718848,-0.530718848,-0.467265989,0.467265989],[0,0,0,0],[9E+09,9E+09,9E+09,9E+09,9E+09,9E+09]];
  CONST robtarget Target_3060:=[[275.51917307,-5.64102153,120],[0.474313597,-0.474313597,-0.524429797,0.524429797],[0,0,0,0],[9E+09,9E+09,9E+09,9E+09,9E+09,9E+09]];
  CONST robtarget Target_3070:=[[273.400942641,4.110051591,120],[0.411790408,-0.411790408,-0.574829244,0.574829244],[0,0,0,0],[9E+09,9E+09,9E+09,9E+09,9E+09,9E+09]];
  CONST robtarget Target_3080:=[[269.140125531,13.133120068,120],[0.343955739,-0.343955739,-0.617814252,0.617814252],[0,0,0,0],[9E+09,9E+09,9E+09,9E+09,9E+09,9E+09]];
  CONST robtarget Target_3090:=[[262.955845572,20.964148645,120],[0.271684554,-0.271684554,-0.652830379,0.652830379],[0,0,0,0],[9E+09,9E+09,9E+09,9E+09,9E+09,9E+09]];
  CONST robtarget Target_3100:=[[255.166145782,27.200405884,120],[0.195909044,-0.195909044,-0.679425968,0.679425968],[0,0,0,0],[9E+09,9E+09,9E+09,9E+09,9E+09,9E+09]];
  CONST robtarget Target_3110:=[[246.171632155,31.521175699,120],[0.117606599,-0.117606599,-0.697257978,0.697257978],[0,0,0,0],[9E+09,9E+09,9E+09,9E+09,9E+09,9E+09]];
  CONST robtarget Target_3120:=[[236.434871438,33.70425103,120],[0.037787206,-0.037787206,-0.706096401,0.706096401],[0,0,0,0],[9E+09,9E+09,9E+09,9E+09,9E+09,9E+09]];
  CONST robtarget Target_3130:=[[226.456602401,33.637361432,120],[0.042519587,-0.042519587,0.705827234,-0.705827234],[0,0,0,0],[9E+09,9E+09,9E+09,9E+09,9E+09,9E+09]];
  CONST robtarget Target_3140:=[[216.749984026,31.323946879,120],[0.12227794,-0.12227794,0.696453951,-0.696453951],[0,0,0,0],[9E+09,9E+09,9E+09,9E+09,9E+09,9E+09]];
  CONST robtarget Target_3150:=[[207.814204935,26.882980857,120],[0.20045909,-0.20045909,0.678097451,-0.678097451],[0,0,0,0],[9E+09,9E+09,9E+09,9E+09,9E+09,9E+09]];
  CONST robtarget Target_3160:=[[200.108811293,20.542851836,120],[0.276054617,-0.276054617,0.650994507,-0.650994507],[0,0,0,0],[9E+09,9E+09,9E+09,9E+09,9E+09,9E+09]];
  CONST robtarget Target_3170:=[[194.030073428,12.629617784,120],[0.348089452,-0.348089452,0.615494706,-0.615494706],[0,0,0,0],[9E+09,9E+09,9E+09,9E+09,9E+09,9E+09]];
  CONST robtarget Target_3180:=[[189.890606575,3.550237775,120],[0.415634453,-0.415634453,0.572055942,-0.572055942],[0,0,0,0],[9E+09,9E+09,9E+09,9E+09,9E+09,9E+09]];
  CONST robtarget Target_3190:=[[187.903293808,-6.228356968,120],[0.47781839,-0.47781839,0.521238511,-0.521238511],[0,0,0,0],[9E+09,9E+09,9E+09,9E+09,9E+09,9E+09]];
  CONST robtarget Target_3200:=[[188.170337963,-16.203276245,120],[0.533839184,-0.533839184,0.463697882,-0.463697882],[0,0,0,0],[9E+09,9E+09,9E+09,9E+09,9E+09,9E+09]];
  CONST robtarget Target_3210:=[[190.678005584,-25.861533349,120],[0.582974249,-0.582974249,0.400176242,-0.400176242],[0,0,0,0],[9E+09,9E+09,9E+09,9E+09,9E+09,9E+09]];
  CONST robtarget Target_3220:=[[195.297333207,-34.706426762,120],[0.624589817,-0.624589817,0.331492927,-0.331492927],[0,0,0,0],[9E+09,9E+09,9E+09,9E+09,9E+09,9E+09]];
  CONST robtarget Target_3230_custom_ends_p2:=[[187.015448949,-40.310924343,120],[0.624589817,-0.624589817,0.331492927,-0.331492927],[0,0,0,0],[9E+09,9E+09,9E+09,9E+09,9E+09,9E+09]];
  CONST robtarget Target_3230:=[[0,260.954122306,130],[0,-0.5,0.866025404,0],[0,0,0,0],[9E+09,9E+09,9E+09,9E+09,9E+09,9E+09]];
  CONST robtarget Target_3240_triangle_starts:=[[0,260.954122306,120],[0,-0.5,0.866025404,0],[0,0,0,0],[9E+09,9E+09,9E+09,9E+09,9E+09,9E+09]];
  CONST robtarget Target_3250:=[[-5,252.293868268,120],[0,-0.5,0.866025404,0],[0,0,0,0],[9E+09,9E+09,9E+09,9E+09,9E+09,9E+09]];
  CONST robtarget Target_3260:=[[-10,243.63361423,120],[0,-0.5,0.866025404,0],[0,0,0,0],[9E+09,9E+09,9E+09,9E+09,9E+09,9E+09]];
  CONST robtarget Target_3270:=[[-15,234.973360192,120],[0,-0.5,0.866025404,0],[0,0,0,0],[9E+09,9E+09,9E+09,9E+09,9E+09,9E+09]];
  CONST robtarget Target_3280:=[[-20,226.313106154,120],[0,-0.5,0.866025404,0],[0,0,0,0],[9E+09,9E+09,9E+09,9E+09,9E+09,9E+09]];
  CONST robtarget Target_3290:=[[-25,217.652852117,120],[0,-0.5,0.866025404,0],[0,0,0,0],[9E+09,9E+09,9E+09,9E+09,9E+09,9E+09]];
  CONST robtarget Target_3300:=[[-30,208.992598079,120],[0,-0.5,0.866025404,0],[0,0,0,0],[9E+09,9E+09,9E+09,9E+09,9E+09,9E+09]];
  CONST robtarget Target_3310:=[[-20,208.992598079,120],[0,1,0,0],[0,0,0,0],[9E+09,9E+09,9E+09,9E+09,9E+09,9E+09]];
  CONST robtarget Target_3320:=[[-10,208.992598079,120],[0,1,0,0],[0,0,0,0],[9E+09,9E+09,9E+09,9E+09,9E+09,9E+09]];
  CONST robtarget Target_3330:=[[0,208.992598079,120],[0,1,0,0],[0,0,0,0],[9E+09,9E+09,9E+09,9E+09,9E+09,9E+09]];
  CONST robtarget Target_3340:=[[10,208.992598079,120],[0,1,0,0],[0,0,0,0],[9E+09,9E+09,9E+09,9E+09,9E+09,9E+09]];
  CONST robtarget Target_3350:=[[20,208.992598079,120],[0,1,0,0],[0,0,0,0],[9E+09,9E+09,9E+09,9E+09,9E+09,9E+09]];
  CONST robtarget Target_3360:=[[30,208.992598079,120],[0,0.5,0.866025404,0],[0,0,0,0],[9E+09,9E+09,9E+09,9E+09,9E+09,9E+09]];
  CONST robtarget Target_3370:=[[25,217.652852117,120],[0,0.5,0.866025404,0],[0,0,0,0],[9E+09,9E+09,9E+09,9E+09,9E+09,9E+09]];
  CONST robtarget Target_3380:=[[20,226.313106154,120],[0,0.5,0.866025404,0],[0,0,0,0],[9E+09,9E+09,9E+09,9E+09,9E+09,9E+09]];
  CONST robtarget Target_3390:=[[15,234.973360192,120],[0,0.5,0.866025404,0],[0,0,0,0],[9E+09,9E+09,9E+09,9E+09,9E+09,9E+09]];
  CONST robtarget Target_3400:=[[10,243.63361423,120],[0,0.5,0.866025404,0],[0,0,0,0],[9E+09,9E+09,9E+09,9E+09,9E+09,9E+09]];
  CONST robtarget Target_3410:=[[5,252.293868268,120],[0,0.5,0.866025404,0],[0,0,0,0],[9E+09,9E+09,9E+09,9E+09,9E+09,9E+09]];
  CONST robtarget Target_3420:=[[0,260.954122306,120],[0,0.5,0.866025404,0],[0,0,0,0],[9E+09,9E+09,9E+09,9E+09,9E+09,9E+09]];
  CONST robtarget Target_3430_triangle_ends:=[[0,260.954122306,130],[0,0.5,0.866025404,0],[0,0,0,0],[9E+09,9E+09,9E+09,9E+09,9E+09,9E+09]];
  CONST robtarget Target_3440_line1_starts:=[[101.66356908,249.31941686,120],[0.590292615,0.590292615,0.389300178,0.389300178],[0,0,0,0],[9E+09,9E+09,9E+09,9E+09,9E+09,9E+09]];
  CONST robtarget Target_3450:=[[110.855609891,245.381602017,120],[0.590292615,0.590292615,0.389300178,0.389300178],[0,0,0,0],[9E+09,9E+09,9E+09,9E+09,9E+09,9E+09]];
  CONST robtarget Target_3460:=[[119.154614128,243.675408233,120],[0,0.979592793,-0.200992436,0],[0,0,0,0],[9E+09,9E+09,9E+09,9E+09,9E+09,9E+09]];
  CONST robtarget Target_3470:=[[128.346654939,239.73759339,120],[0,0.979592793,-0.200992436,0],[0,0,0,0],[9E+09,9E+09,9E+09,9E+09,9E+09,9E+09]];
  CONST robtarget Target_3480:=[[137.53869575,235.799778548,120],[0,0.979592793,-0.200992436,0],[0,0,0,0],[9E+09,9E+09,9E+09,9E+09,9E+09,9E+09]];
  CONST robtarget Target_3490:=[[146.730736561,231.861963706,120],[0,0.979592793,-0.200992436,0],[0,0,0,0],[9E+09,9E+09,9E+09,9E+09,9E+09,9E+09]];
  CONST robtarget Target_3500:=[[155.922777371,227.924148864,120],[0,0.979592793,-0.200992436,0],[0,0,0,0],[9E+09,9E+09,9E+09,9E+09,9E+09,9E+09]];
  CONST robtarget Target_3510:=[[165.114818182,223.986334022,120],[0,0.979592793,-0.200992436,0],[0,0,0,0],[9E+09,9E+09,9E+09,9E+09,9E+09,9E+09]];
  CONST robtarget Target_3520:=[[159.152373975,224.691559583,120],[0,0.979592793,-0.200992436,0],[0,0,0,0],[9E+09,9E+09,9E+09,9E+09,9E+09,9E+09]];
  CONST robtarget Target_3530:=[[149.960333164,228.629374425,120],[0,0.979592793,-0.200992436,0],[0,0,0,0],[9E+09,9E+09,9E+09,9E+09,9E+09,9E+09]];
  CONST robtarget Target_3540:=[[140.768292353,232.567189267,120],[0,0.979592793,-0.200992436,0],[0,0,0,0],[9E+09,9E+09,9E+09,9E+09,9E+09,9E+09]];
  CONST robtarget Target_3550:=[[131.576251542,236.505004109,120],[0,0.979592793,-0.200992436,0],[0,0,0,0],[9E+09,9E+09,9E+09,9E+09,9E+09,9E+09]];
  CONST robtarget Target_3560:=[[122.384210731,240.442818952,120],[0,0.979592793,-0.200992436,0],[0,0,0,0],[9E+09,9E+09,9E+09,9E+09,9E+09,9E+09]];
  CONST robtarget Target_3570:=[[113.19216992,244.380633794,120],[0,0.979592793,-0.200992436,0],[0,0,0,0],[9E+09,9E+09,9E+09,9E+09,9E+09,9E+09]];
  CONST robtarget Target_3580_line1_ends:=[[113.19216992,244.380633794,130],[0,0.979592793,-0.200992436,0],[0,0,0,0],[9E+09,9E+09,9E+09,9E+09,9E+09,9E+09]];
  CONST robtarget Target_3590_line2_starts:=[[89.9320837,225.555374256,120],[0.590292615,0.590292615,0.389300178,0.389300178],[0,0,0,0],[9E+09,9E+09,9E+09,9E+09,9E+09,9E+09]];
  CONST robtarget Target_3600:=[[99.124124511,221.617559414,120],[0.590292615,0.590292615,0.389300178,0.389300178],[0,0,0,0],[9E+09,9E+09,9E+09,9E+09,9E+09,9E+09]];
  CONST robtarget Target_3610:=[[107.423128748,219.911365629,120],[0,0.979592793,-0.200992436,0],[0,0,0,0],[9E+09,9E+09,9E+09,9E+09,9E+09,9E+09]];
  CONST robtarget Target_3620:=[[116.615169559,215.973550787,120],[0,0.979592793,-0.200992436,0],[0,0,0,0],[9E+09,9E+09,9E+09,9E+09,9E+09,9E+09]];
  CONST robtarget Target_3630:=[[125.80721037,212.035735945,120],[0,0.979592793,-0.200992436,0],[0,0,0,0],[9E+09,9E+09,9E+09,9E+09,9E+09,9E+09]];
  CONST robtarget Target_3640:=[[134.999251181,208.097921103,120],[0,0.979592793,-0.200992436,0],[0,0,0,0],[9E+09,9E+09,9E+09,9E+09,9E+09,9E+09]];
  CONST robtarget Target_3650:=[[144.191291991,204.160106261,120],[0,0.979592793,-0.200992436,0],[0,0,0,0],[9E+09,9E+09,9E+09,9E+09,9E+09,9E+09]];
  CONST robtarget Target_3660:=[[153.383332802,200.222291419,120],[0,0.979592793,-0.200992436,0],[0,0,0,0],[9E+09,9E+09,9E+09,9E+09,9E+09,9E+09]];
  CONST robtarget Target_3670:=[[147.420888595,200.92751698,120],[0,0.979592793,-0.200992436,0],[0,0,0,0],[9E+09,9E+09,9E+09,9E+09,9E+09,9E+09]];
  CONST robtarget Target_3680:=[[138.228847784,204.865331822,120],[0,0.979592793,-0.200992436,0],[0,0,0,0],[9E+09,9E+09,9E+09,9E+09,9E+09,9E+09]];
  CONST robtarget Target_3690:=[[129.036806973,208.803146664,120],[0,0.979592793,-0.200992436,0],[0,0,0,0],[9E+09,9E+09,9E+09,9E+09,9E+09,9E+09]];
  CONST robtarget Target_3700:=[[119.844766162,212.740961506,120],[0,0.979592793,-0.200992436,0],[0,0,0,0],[9E+09,9E+09,9E+09,9E+09,9E+09,9E+09]];
  CONST robtarget Target_3710:=[[110.652725351,216.678776348,120],[0,0.979592793,-0.200992436,0],[0,0,0,0],[9E+09,9E+09,9E+09,9E+09,9E+09,9E+09]];
  CONST robtarget Target_3720:=[[101.46068454,220.616591191,120],[0,0.979592793,-0.200992436,0],[0,0,0,0],[9E+09,9E+09,9E+09,9E+09,9E+09,9E+09]];
  CONST robtarget Target_3730_line2_ends:=[[101.46068454,220.616591191,130],[0,0.979592793,-0.200992436,0],[0,0,0,0],[9E+09,9E+09,9E+09,9E+09,9E+09,9E+09]];
  CONST robtarget Target_3740_line3_starts:=[[78.948458053,197.771331126,120],[0.590292615,0.590292615,0.389300178,0.389300178],[0,0,0,0],[9E+09,9E+09,9E+09,9E+09,9E+09,9E+09]];
  CONST robtarget Target_3750:=[[88.140498864,193.833516284,120],[0.590292615,0.590292615,0.389300178,0.389300178],[0,0,0,0],[9E+09,9E+09,9E+09,9E+09,9E+09,9E+09]];
  CONST robtarget Target_3760:=[[96.439503101,192.127322499,120],[0,0.979592793,-0.200992436,0],[0,0,0,0],[9E+09,9E+09,9E+09,9E+09,9E+09,9E+09]];
  CONST robtarget Target_3770:=[[105.631543912,188.189507657,120],[0,0.979592793,-0.200992436,0],[0,0,0,0],[9E+09,9E+09,9E+09,9E+09,9E+09,9E+09]];
  CONST robtarget Target_3780:=[[114.823584722,184.251692815,120],[0,0.979592793,-0.200992436,0],[0,0,0,0],[9E+09,9E+09,9E+09,9E+09,9E+09,9E+09]];
  CONST robtarget Target_3790:=[[124.015625533,180.313877972,120],[0,0.979592793,-0.200992436,0],[0,0,0,0],[9E+09,9E+09,9E+09,9E+09,9E+09,9E+09]];
  CONST robtarget Target_3800:=[[133.207666344,176.37606313,120],[0,0.979592793,-0.200992436,0],[0,0,0,0],[9E+09,9E+09,9E+09,9E+09,9E+09,9E+09]];
  CONST robtarget Target_3810:=[[142.399707155,172.438248288,120],[0,0.979592793,-0.200992436,0],[0,0,0,0],[9E+09,9E+09,9E+09,9E+09,9E+09,9E+09]];
  CONST robtarget Target_3820:=[[136.437262948,173.143473849,120],[0,0.979592793,-0.200992436,0],[0,0,0,0],[9E+09,9E+09,9E+09,9E+09,9E+09,9E+09]];
  CONST robtarget Target_3830:=[[127.245222137,177.081288691,120],[0,0.979592793,-0.200992436,0],[0,0,0,0],[9E+09,9E+09,9E+09,9E+09,9E+09,9E+09]];
  CONST robtarget Target_3840:=[[118.053181326,181.019103534,120],[0,0.979592793,-0.200992436,0],[0,0,0,0],[9E+09,9E+09,9E+09,9E+09,9E+09,9E+09]];
  CONST robtarget Target_3850:=[[108.861140515,184.956918376,120],[0,0.979592793,-0.200992436,0],[0,0,0,0],[9E+09,9E+09,9E+09,9E+09,9E+09,9E+09]];
  CONST robtarget Target_3860:=[[99.669099704,188.894733218,120],[0,0.979592793,-0.200992436,0],[0,0,0,0],[9E+09,9E+09,9E+09,9E+09,9E+09,9E+09]];
  CONST robtarget Target_3870:=[[90.477058893,192.83254806,120],[0,0.979592793,-0.200992436,0],[0,0,0,0],[9E+09,9E+09,9E+09,9E+09,9E+09,9E+09]];
  CONST robtarget Target_3880_line3_ends:=[[90.477058893,192.83254806,130],[0,0.979592793,-0.200992436,0],[0,0,0,0],[9E+09,9E+09,9E+09,9E+09,9E+09,9E+09]];
  PROC Path_10()
  ENDPROC
  PROC Path_20()
    MoveL Target_80_outter_ring_starts,v1000,z100,ToolM_DS109\WObj:=Workobject_2;
    MoveL Target_90,v1000,z100,ToolM_DS109\WObj:=Workobject_2;
    MoveL Target_100,v1000,z100,ToolM_DS109\WObj:=Workobject_2;
    MoveL Target_110,v1000,z100,ToolM_DS109\WObj:=Workobject_2;
    MoveL Target_120,v1000,z100,ToolM_DS109\WObj:=Workobject_2;
    MoveL Target_130,v1000,z100,ToolM_DS109\WObj:=Workobject_2;
    MoveL Target_140,v1000,z100,ToolM_DS109\WObj:=Workobject_2;
    MoveL Target_150,v1000,z100,ToolM_DS109\WObj:=Workobject_2;
    MoveL Target_160,v1000,z100,ToolM_DS109\WObj:=Workobject_2;
    MoveL Target_170,v1000,z100,ToolM_DS109\WObj:=Workobject_2;
    MoveL Target_180,v1000,z100,ToolM_DS109\WObj:=Workobject_2;
    MoveL Target_190,v1000,z100,ToolM_DS109\WObj:=Workobject_2;
    MoveL Target_200,v1000,z100,ToolM_DS109\WObj:=Workobject_2;
    MoveL Target_210,v1000,z100,ToolM_DS109\WObj:=Workobject_2;
    MoveL Target_220,v1000,z100,ToolM_DS109\WObj:=Workobject_2;
    MoveL Target_230,v1000,z100,ToolM_DS109\WObj:=Workobject_2;
    MoveL Target_240,v1000,z100,ToolM_DS109\WObj:=Workobject_2;
    MoveL Target_250,v1000,z100,ToolM_DS109\WObj:=Workobject_2;
    MoveL Target_260,v1000,z100,ToolM_DS109\WObj:=Workobject_2;
    MoveL Target_270,v1000,z100,ToolM_DS109\WObj:=Workobject_2;
    MoveL Target_280_outter_ring_half,v1000,z100,ToolM_DS109\WObj:=Workobject_2;
    MoveL Target_290,v1000,z100,ToolM_DS109\WObj:=Workobject_2;
    MoveL Target_300,v1000,z100,ToolM_DS109\WObj:=Workobject_2;
    MoveL Target_310,v1000,z100,ToolM_DS109\WObj:=Workobject_2;
    MoveL Target_320,v1000,z100,ToolM_DS109\WObj:=Workobject_2;
    MoveL Target_330,v1000,z100,ToolM_DS109\WObj:=Workobject_2;
    MoveL Target_340,v1000,z100,ToolM_DS109\WObj:=Workobject_2;
    MoveL Target_350,v1000,z100,ToolM_DS109\WObj:=Workobject_2;
    MoveL Target_360,v1000,z100,ToolM_DS109\WObj:=Workobject_2;
    MoveL Target_370,v1000,z100,ToolM_DS109\WObj:=Workobject_2;
    MoveL Target_380,v1000,z100,ToolM_DS109\WObj:=Workobject_2;
    MoveL Target_390,v1000,z100,ToolM_DS109\WObj:=Workobject_2;
    MoveL Target_400,v1000,z100,ToolM_DS109\WObj:=Workobject_2;
    MoveL Target_410,v1000,z100,ToolM_DS109\WObj:=Workobject_2;
    MoveL Target_420,v1000,z100,ToolM_DS109\WObj:=Workobject_2;
    MoveL Target_430,v1000,z100,ToolM_DS109\WObj:=Workobject_2;
    MoveL Target_440,v1000,z100,ToolM_DS109\WObj:=Workobject_2;
    MoveL Target_450,v1000,z100,ToolM_DS109\WObj:=Workobject_2;
    MoveL Target_460,v1000,z100,ToolM_DS109\WObj:=Workobject_2;
    MoveL Target_470,v1000,z100,ToolM_DS109\WObj:=Workobject_2;
    MoveL Target_480,v1000,z100,ToolM_DS109\WObj:=Workobject_2;
    MoveL Target_490_outer_ring_ends,v1000,z100,ToolM_DS109\WObj:=Workobject_2;
  ENDPROC
  PROC Path_30()
    MoveL Target_500_inner_ring_starts,v1000,z100,ToolM_DS109\WObj:=Workobject_2;
    MoveL Target_510,v1000,z100,ToolM_DS109\WObj:=Workobject_2;
    MoveL Target_520,v1000,z100,ToolM_DS109\WObj:=Workobject_2;
    MoveL Target_530,v1000,z100,ToolM_DS109\WObj:=Workobject_2;
    MoveL Target_540,v1000,z100,ToolM_DS109\WObj:=Workobject_2;
    MoveL Target_550,v1000,z100,ToolM_DS109\WObj:=Workobject_2;
    MoveL Target_560,v1000,z100,ToolM_DS109\WObj:=Workobject_2;
    MoveL Target_570,v1000,z100,ToolM_DS109\WObj:=Workobject_2;
    MoveL Target_580,v1000,z100,ToolM_DS109\WObj:=Workobject_2;
    MoveL Target_590,v1000,z100,ToolM_DS109\WObj:=Workobject_2;
    MoveL Target_600,v1000,z100,ToolM_DS109\WObj:=Workobject_2;
    MoveL Target_610,v1000,z100,ToolM_DS109\WObj:=Workobject_2;
    MoveL Target_620,v1000,z100,ToolM_DS109\WObj:=Workobject_2;
    MoveL Target_630,v1000,z100,ToolM_DS109\WObj:=Workobject_2;
    MoveL Target_640,v1000,z100,ToolM_DS109\WObj:=Workobject_2;
    MoveL Target_650_inner_ring_half,v1000,z100,ToolM_DS109\WObj:=Workobject_2;
    MoveL Target_660,v1000,z100,ToolM_DS109\WObj:=Workobject_2;
    MoveL Target_670,v1000,z100,ToolM_DS109\WObj:=Workobject_2;
    MoveL Target_680,v1000,z100,ToolM_DS109\WObj:=Workobject_2;
    MoveL Target_690,v1000,z100,ToolM_DS109\WObj:=Workobject_2;
    MoveL Target_700,v1000,z100,ToolM_DS109\WObj:=Workobject_2;
    MoveL Target_710,v1000,z100,ToolM_DS109\WObj:=Workobject_2;
    MoveL Target_720,v1000,z100,ToolM_DS109\WObj:=Workobject_2;
    MoveL Target_730,v1000,z100,ToolM_DS109\WObj:=Workobject_2;
    MoveL Target_740,v1000,z100,ToolM_DS109\WObj:=Workobject_2;
    MoveL Target_750,v1000,z100,ToolM_DS109\WObj:=Workobject_2;
    MoveL Target_760,v1000,z100,ToolM_DS109\WObj:=Workobject_2;
    MoveL Target_770,v1000,z100,ToolM_DS109\WObj:=Workobject_2;
    MoveL Target_780,v1000,z100,ToolM_DS109\WObj:=Workobject_2;
    MoveL Target_790,v1000,z100,ToolM_DS109\WObj:=Workobject_2;
    MoveL Target_800,v1000,z100,ToolM_DS109\WObj:=Workobject_2;
    MoveL Target_810_inner_ring_ends,v1000,z100,ToolM_DS109\WObj:=Workobject_2;
  ENDPROC
  PROC Path_40()
    MoveL Target_810,v1000,z100,ToolM_DS109\WObj:=Workobject_2;
    MoveL Target_820_d_inner_starts,v1000,z100,ToolM_DS109\WObj:=Workobject_2;
    MoveL Target_830,v1000,z100,ToolM_DS109\WObj:=Workobject_2;
    MoveL Target_840,v1000,z100,ToolM_DS109\WObj:=Workobject_2;
    MoveL Target_850,v1000,z100,ToolM_DS109\WObj:=Workobject_2;
    MoveL Target_860,v1000,z100,ToolM_DS109\WObj:=Workobject_2;
    MoveL Target_870,v1000,z100,ToolM_DS109\WObj:=Workobject_2;
    MoveL Target_880,v1000,z100,ToolM_DS109\WObj:=Workobject_2;
    MoveL Target_890,v1000,z100,ToolM_DS109\WObj:=Workobject_2;
    MoveL Target_900,v1000,z100,ToolM_DS109\WObj:=Workobject_2;
    MoveL Target_910,v1000,z100,ToolM_DS109\WObj:=Workobject_2;
    MoveL Target_920,v1000,z100,ToolM_DS109\WObj:=Workobject_2;
    MoveL Target_930,v1000,z100,ToolM_DS109\WObj:=Workobject_2;
    MoveL Target_940_d_inner,v1000,z100,ToolM_DS109\WObj:=Workobject_2;
  ENDPROC
  PROC Path_50()
    MoveL Target_940,v1000,z100,ToolM_DS109\WObj:=Workobject_2;
    MoveL Target_950_d_outter_starts,v1000,z100,ToolM_DS109\WObj:=Workobject_2;
    MoveL Target_960,v1000,z100,ToolM_DS109\WObj:=Workobject_2;
    MoveL Target_970,v1000,z100,ToolM_DS109\WObj:=Workobject_2;
    MoveL Target_980,v1000,z100,ToolM_DS109\WObj:=Workobject_2;
    MoveL Target_990,v1000,z100,ToolM_DS109\WObj:=Workobject_2;
    MoveL Target_1000,v1000,z100,ToolM_DS109\WObj:=Workobject_2;
    MoveL Target_1010,v1000,z100,ToolM_DS109\WObj:=Workobject_2;
    MoveL Target_1020,v1000,z100,ToolM_DS109\WObj:=Workobject_2;
    MoveL Target_1030,v1000,z100,ToolM_DS109\WObj:=Workobject_2;
    MoveL Target_1040,v1000,z100,ToolM_DS109\WObj:=Workobject_2;
    MoveL Target_1050,v1000,z100,ToolM_DS109\WObj:=Workobject_2;
    MoveL Target_1060,v1000,z100,ToolM_DS109\WObj:=Workobject_2;
    MoveL Target_1070_d_outter_ends,v1000,z100,ToolM_DS109\WObj:=Workobject_2;
  ENDPROC
  PROC Path_60()
    MoveL Target_1070,v1000,z100,ToolM_DS109\WObj:=Workobject_2;
    MoveL Target_1080_s_starts,v1000,z100,ToolM_DS109\WObj:=Workobject_2;
    MoveL Target_1090,v1000,z100,ToolM_DS109\WObj:=Workobject_2;
    MoveL Target_1100,v1000,z100,ToolM_DS109\WObj:=Workobject_2;
    MoveL Target_1110,v1000,z100,ToolM_DS109\WObj:=Workobject_2;
    MoveL Target_1120,v1000,z100,ToolM_DS109\WObj:=Workobject_2;
    MoveL Target_1130,v1000,z100,ToolM_DS109\WObj:=Workobject_2;
    MoveL Target_1140,v1000,z100,ToolM_DS109\WObj:=Workobject_2;
    MoveL Target_1150,v1000,z100,ToolM_DS109\WObj:=Workobject_2;
    MoveL Target_1160,v1000,z100,ToolM_DS109\WObj:=Workobject_2;
    MoveL Target_1170,v1000,z100,ToolM_DS109\WObj:=Workobject_2;
    MoveL Target_1180,v1000,z100,ToolM_DS109\WObj:=Workobject_2;
    MoveL Target_1190,v1000,z100,ToolM_DS109\WObj:=Workobject_2;
    MoveL Target_1200,v1000,z100,ToolM_DS109\WObj:=Workobject_2;
    MoveL Target_1210,v1000,z100,ToolM_DS109\WObj:=Workobject_2;
    MoveL Target_1220,v1000,z100,ToolM_DS109\WObj:=Workobject_2;
    MoveL Target_1230,v1000,z100,ToolM_DS109\WObj:=Workobject_2;
    MoveL Target_1240,v1000,z100,ToolM_DS109\WObj:=Workobject_2;
    MoveL Target_1250,v1000,z100,ToolM_DS109\WObj:=Workobject_2;
    MoveL Target_1260,v1000,z100,ToolM_DS109\WObj:=Workobject_2;
    MoveL Target_1270,v1000,z100,ToolM_DS109\WObj:=Workobject_2;
    MoveL Target_1280,v1000,z100,ToolM_DS109\WObj:=Workobject_2;
    MoveL Target_1290,v1000,z100,ToolM_DS109\WObj:=Workobject_2;
    MoveL Target_1300,v1000,z100,ToolM_DS109\WObj:=Workobject_2;
    MoveL Target_1310,v1000,z100,ToolM_DS109\WObj:=Workobject_2;
    MoveL Target_1320,v1000,z100,ToolM_DS109\WObj:=Workobject_2;
    MoveL Target_1330,v1000,z100,ToolM_DS109\WObj:=Workobject_2;
    MoveL Target_1340,v1000,z100,ToolM_DS109\WObj:=Workobject_2;
    MoveL Target_1350,v1000,z100,ToolM_DS109\WObj:=Workobject_2;
    MoveL Target_1360,v1000,z100,ToolM_DS109\WObj:=Workobject_2;
    MoveL Target_1370,v1000,z100,ToolM_DS109\WObj:=Workobject_2;
    MoveL Target_1380,v1000,z100,ToolM_DS109\WObj:=Workobject_2;
    MoveL Target_1390,v1000,z100,ToolM_DS109\WObj:=Workobject_2;
    MoveL Target_1400,v1000,z100,ToolM_DS109\WObj:=Workobject_2;
    MoveL Target_1410,v1000,z100,ToolM_DS109\WObj:=Workobject_2;
    MoveL Target_1420,v1000,z100,ToolM_DS109\WObj:=Workobject_2;
    MoveL Target_1430,v1000,z100,ToolM_DS109\WObj:=Workobject_2;
    MoveL Target_1440_s_ends,v1000,z100,ToolM_DS109\WObj:=Workobject_2;
  ENDPROC
  PROC Path_70()
    MoveL Target_1440,v1000,z100,ToolM_DS109\WObj:=Workobject_2;
    MoveL Target_1450_circle_starts,v1000,z100,ToolM_DS109\WObj:=Workobject_2;
    MoveL Target_1460,v1000,z100,ToolM_DS109\WObj:=Workobject_2;
    MoveL Target_1470,v1000,z100,ToolM_DS109\WObj:=Workobject_2;
    MoveL Target_1480,v1000,z100,ToolM_DS109\WObj:=Workobject_2;
    MoveL Target_1490,v1000,z100,ToolM_DS109\WObj:=Workobject_2;
    MoveL Target_1500,v1000,z100,ToolM_DS109\WObj:=Workobject_2;
    MoveL Target_1510,v1000,z100,ToolM_DS109\WObj:=Workobject_2;
    MoveL Target_1520,v1000,z100,ToolM_DS109\WObj:=Workobject_2;
    MoveL Target_1530,v1000,z100,ToolM_DS109\WObj:=Workobject_2;
    MoveL Target_1540,v1000,z100,ToolM_DS109\WObj:=Workobject_2;
    MoveL Target_1550,v1000,z100,ToolM_DS109\WObj:=Workobject_2;
    MoveL Target_1560,v1000,z100,ToolM_DS109\WObj:=Workobject_2;
    MoveL Target_1570,v1000,z100,ToolM_DS109\WObj:=Workobject_2;
    MoveL Target_1580,v1000,z100,ToolM_DS109\WObj:=Workobject_2;
    MoveL Target_1590,v1000,z100,ToolM_DS109\WObj:=Workobject_2;
    MoveL Target_1600_circle_ends,v1000,z100,ToolM_DS109\WObj:=Workobject_2;
  ENDPROC
  PROC Path_80()
  ENDPROC
  PROC Path_90()
  ENDPROC
  PROC Path_100()
    MoveC Target_2450_point1_starts,Target_2460,v1000,z100,ToolM_DS109\WObj:=Workobject_2;
    MoveC Target_2470,Target_2480_point1_ends,v1000,z100,ToolM_DS109\WObj:=Workobject_2;
  ENDPROC
  PROC Path_110()
    MoveL Target_2480,v1000,z100,ToolM_DS109\WObj:=Workobject_2;
    MoveL Target_2490_point2_starts,v1000,z100,ToolM_DS109\WObj:=Workobject_2;
    MoveC Target_2500,Target_2510,v1000,z100,ToolM_DS109\WObj:=Workobject_2;
    MoveC Target_2520,Target_2530,v1000,z100,ToolM_DS109\WObj:=Workobject_2;
    MoveL Target_2540_point2_ends,v1000,z100,ToolM_DS109\WObj:=Workobject_2;
  ENDPROC
  PROC Path_120()
    MoveL Target_2540,v1000,z100,ToolM_DS109\WObj:=Workobject_2;
    MoveL Target_2550_point3_starts,v1000,z100,ToolM_DS109\WObj:=Workobject_2;
    MoveC Target_2560,Target_2570,v1000,z100,ToolM_DS109\WObj:=Workobject_2;
    MoveC Target_2580,Target_2590,v1000,z100,ToolM_DS109\WObj:=Workobject_2;
    MoveL Target_2600_point3_ends,v1000,z100,ToolM_DS109\WObj:=Workobject_2;
  ENDPROC
  PROC Path_130()
    MoveL Target_2600,v1000,z100,ToolM_DS109\WObj:=Workobject_2;
    MoveL Target_2610_point4_starts,v1000,z100,ToolM_DS109\WObj:=Workobject_2;
    MoveC Target_2620,Target_2630,v1000,z100,ToolM_DS109\WObj:=Workobject_2;
    MoveC Target_2640,Target_2650,v1000,z100,ToolM_DS109\WObj:=Workobject_2;
    MoveL Target_2660_point4_ends,v1000,z100,ToolM_DS109\WObj:=Workobject_2;
  ENDPROC
  PROC Path_140()
    MoveL Target_2660,v1000,z100,ToolM_DS109\WObj:=Workobject_2;
    MoveL Target_2670_point5_starts,v1000,z100,ToolM_DS109\WObj:=Workobject_2;
    MoveC Target_2680,Target_2690,v1000,z100,ToolM_DS109\WObj:=Workobject_2;
    MoveC Target_2700,Target_2710,v1000,z100,ToolM_DS109\WObj:=Workobject_2;
    MoveL Target_2720_point5_ends,v1000,z100,ToolM_DS109\WObj:=Workobject_2;
  ENDPROC
  PROC Path_150()
    MoveL Target_2720,v1000,z100,ToolM_DS109\WObj:=Workobject_2;
    MoveL Target_2730_custom_starts_p1,v1000,z100,ToolM_DS109\WObj:=Workobject_2;
    MoveL Target_2740,v1000,z100,ToolM_DS109\WObj:=Workobject_2;
    MoveL Target_2750,v1000,z100,ToolM_DS109\WObj:=Workobject_2;
    MoveL Target_2760,v1000,z100,ToolM_DS109\WObj:=Workobject_2;
    MoveL Target_2770,v1000,z100,ToolM_DS109\WObj:=Workobject_2;
    MoveL Target_2780,v1000,z100,ToolM_DS109\WObj:=Workobject_2;
    MoveL Target_2790,v1000,z100,ToolM_DS109\WObj:=Workobject_2;
    MoveL Target_2800,v1000,z100,ToolM_DS109\WObj:=Workobject_2;
    MoveL Target_2810,v1000,z100,ToolM_DS109\WObj:=Workobject_2;
    MoveL Target_2820,v1000,z100,ToolM_DS109\WObj:=Workobject_2;
    MoveL Target_2830,v1000,z100,ToolM_DS109\WObj:=Workobject_2;
    MoveL Target_2840,v1000,z100,ToolM_DS109\WObj:=Workobject_2;
    MoveL Target_2850,v1000,z100,ToolM_DS109\WObj:=Workobject_2;
    MoveL Target_2860,v1000,z100,ToolM_DS109\WObj:=Workobject_2;
    MoveL Target_2870,v1000,z100,ToolM_DS109\WObj:=Workobject_2;
    MoveL Target_2880,v1000,z100,ToolM_DS109\WObj:=Workobject_2;
    MoveL Target_2890,v1000,z100,ToolM_DS109\WObj:=Workobject_2;
    MoveL Target_2900,v1000,z100,ToolM_DS109\WObj:=Workobject_2;
    MoveL Target_2910,v1000,z100,ToolM_DS109\WObj:=Workobject_2;
    MoveL Target_2920,v1000,z100,ToolM_DS109\WObj:=Workobject_2;
    MoveL Target_2930,v1000,z100,ToolM_DS109\WObj:=Workobject_2;
    MoveL Target_2940_custom_ends_p1,v1000,z100,ToolM_DS109\WObj:=Workobject_2;
  ENDPROC
  PROC Path_160()
    MoveL Target_2940,v1000,z100,ToolM_DS109\WObj:=Workobject_2;
    MoveL Target_2950_custom_start_p1,v1000,z100,ToolM_DS109\WObj:=Workobject_2;
    MoveL Target_2960,v1000,z100,ToolM_DS109\WObj:=Workobject_2;
    MoveL Target_2970,v1000,z100,ToolM_DS109\WObj:=Workobject_2;
    MoveL Target_2980,v1000,z100,ToolM_DS109\WObj:=Workobject_2;
    MoveL Target_2990,v1000,z100,ToolM_DS109\WObj:=Workobject_2;
    MoveL Target_3000,v1000,z100,ToolM_DS109\WObj:=Workobject_2;
    MoveL Target_3010,v1000,z100,ToolM_DS109\WObj:=Workobject_2;
    MoveL Target_3020,v1000,z100,ToolM_DS109\WObj:=Workobject_2;
    MoveL Target_3030,v1000,z100,ToolM_DS109\WObj:=Workobject_2;
    MoveL Target_3040,v1000,z100,ToolM_DS109\WObj:=Workobject_2;
    MoveL Target_3050,v1000,z100,ToolM_DS109\WObj:=Workobject_2;
    MoveL Target_3060,v1000,z100,ToolM_DS109\WObj:=Workobject_2;
    MoveL Target_3070,v1000,z100,ToolM_DS109\WObj:=Workobject_2;
    MoveL Target_3080,v1000,z100,ToolM_DS109\WObj:=Workobject_2;
    MoveL Target_3090,v1000,z100,ToolM_DS109\WObj:=Workobject_2;
    MoveL Target_3100,v1000,z100,ToolM_DS109\WObj:=Workobject_2;
    MoveL Target_3110,v1000,z100,ToolM_DS109\WObj:=Workobject_2;
    MoveL Target_3120,v1000,z100,ToolM_DS109\WObj:=Workobject_2;
    MoveL Target_3130,v1000,z100,ToolM_DS109\WObj:=Workobject_2;
    MoveL Target_3140,v1000,z100,ToolM_DS109\WObj:=Workobject_2;
    MoveL Target_3150,v1000,z100,ToolM_DS109\WObj:=Workobject_2;
    MoveL Target_3160,v1000,z100,ToolM_DS109\WObj:=Workobject_2;
    MoveL Target_3170,v1000,z100,ToolM_DS109\WObj:=Workobject_2;
    MoveL Target_3180,v1000,z100,ToolM_DS109\WObj:=Workobject_2;
    MoveL Target_3190,v1000,z100,ToolM_DS109\WObj:=Workobject_2;
    MoveL Target_3200,v1000,z100,ToolM_DS109\WObj:=Workobject_2;
    MoveL Target_3210,v1000,z100,ToolM_DS109\WObj:=Workobject_2;
    MoveL Target_3220,v1000,z100,ToolM_DS109\WObj:=Workobject_2;
    MoveL Target_3230_custom_ends_p2,v1000,z100,ToolM_DS109\WObj:=Workobject_2;
  ENDPROC
  PROC Path_170()
    MoveL Target_3230,v1000,z100,ToolM_DS109\WObj:=Workobject_2;
    MoveL Target_3240_triangle_starts,v1000,z100,ToolM_DS109\WObj:=Workobject_2;
    MoveL Target_3250,v1000,z100,ToolM_DS109\WObj:=Workobject_2;
    MoveL Target_3260,v1000,z100,ToolM_DS109\WObj:=Workobject_2;
    MoveL Target_3270,v1000,z100,ToolM_DS109\WObj:=Workobject_2;
    MoveL Target_3280,v1000,z100,ToolM_DS109\WObj:=Workobject_2;
    MoveL Target_3290,v1000,z100,ToolM_DS109\WObj:=Workobject_2;
    MoveL Target_3300,v1000,z100,ToolM_DS109\WObj:=Workobject_2;
    MoveL Target_3310,v1000,z100,ToolM_DS109\WObj:=Workobject_2;
    MoveL Target_3320,v1000,z100,ToolM_DS109\WObj:=Workobject_2;
    MoveL Target_3330,v1000,z100,ToolM_DS109\WObj:=Workobject_2;
    MoveL Target_3340,v1000,z100,ToolM_DS109\WObj:=Workobject_2;
    MoveL Target_3350,v1000,z100,ToolM_DS109\WObj:=Workobject_2;
    MoveL Target_3360,v1000,z100,ToolM_DS109\WObj:=Workobject_2;
    MoveL Target_3370,v1000,z100,ToolM_DS109\WObj:=Workobject_2;
    MoveL Target_3380,v1000,z100,ToolM_DS109\WObj:=Workobject_2;
    MoveL Target_3390,v1000,z100,ToolM_DS109\WObj:=Workobject_2;
    MoveL Target_3400,v1000,z100,ToolM_DS109\WObj:=Workobject_2;
    MoveL Target_3410,v1000,z100,ToolM_DS109\WObj:=Workobject_2;
    MoveL Target_3420,v1000,z100,ToolM_DS109\WObj:=Workobject_2;
    MoveL Target_3430_triangle_ends,v1000,z100,ToolM_DS109\WObj:=Workobject_2;
  ENDPROC
  PROC Path_180()
  ENDPROC
  PROC Path_190()
  ENDPROC
  PROC Path_200()
    MoveL Target_3440_line1_starts,v1000,z100,ToolM_DS109\WObj:=Workobject_2;
    MoveL Target_3450,v1000,z100,ToolM_DS109\WObj:=Workobject_2;
    MoveL Target_3460,v1000,z100,ToolM_DS109\WObj:=Workobject_2;
    MoveL Target_3470,v1000,z100,ToolM_DS109\WObj:=Workobject_2;
    MoveL Target_3480,v1000,z100,ToolM_DS109\WObj:=Workobject_2;
    MoveL Target_3490,v1000,z100,ToolM_DS109\WObj:=Workobject_2;
    MoveL Target_3500,v1000,z100,ToolM_DS109\WObj:=Workobject_2;
    MoveL Target_3510,v1000,z100,ToolM_DS109\WObj:=Workobject_2;
    MoveL Target_3520,v1000,z100,ToolM_DS109\WObj:=Workobject_2;
    MoveL Target_3530,v1000,z100,ToolM_DS109\WObj:=Workobject_2;
    MoveL Target_3540,v1000,z100,ToolM_DS109\WObj:=Workobject_2;
    MoveL Target_3550,v1000,z100,ToolM_DS109\WObj:=Workobject_2;
    MoveL Target_3560,v1000,z100,ToolM_DS109\WObj:=Workobject_2;
    MoveL Target_3570,v1000,z100,ToolM_DS109\WObj:=Workobject_2;
    MoveL Target_3580_line1_ends,v1000,z100,ToolM_DS109\WObj:=Workobject_2;
  ENDPROC
  PROC Path_210()
    MoveL Target_3590_line2_starts,v1000,z100,ToolM_DS109\WObj:=Workobject_2;
    MoveL Target_3600,v1000,z100,ToolM_DS109\WObj:=Workobject_2;
    MoveL Target_3610,v1000,z100,ToolM_DS109\WObj:=Workobject_2;
    MoveL Target_3620,v1000,z100,ToolM_DS109\WObj:=Workobject_2;
    MoveL Target_3630,v1000,z100,ToolM_DS109\WObj:=Workobject_2;
    MoveL Target_3640,v1000,z100,ToolM_DS109\WObj:=Workobject_2;
    MoveL Target_3650,v1000,z100,ToolM_DS109\WObj:=Workobject_2;
    MoveL Target_3660,v1000,z100,ToolM_DS109\WObj:=Workobject_2;
    MoveL Target_3670,v1000,z100,ToolM_DS109\WObj:=Workobject_2;
    MoveL Target_3680,v1000,z100,ToolM_DS109\WObj:=Workobject_2;
    MoveL Target_3690,v1000,z100,ToolM_DS109\WObj:=Workobject_2;
    MoveL Target_3700,v1000,z100,ToolM_DS109\WObj:=Workobject_2;
    MoveL Target_3710,v1000,z100,ToolM_DS109\WObj:=Workobject_2;
    MoveL Target_3720,v1000,z100,ToolM_DS109\WObj:=Workobject_2;
    MoveL Target_3730_line2_ends,v1000,z100,ToolM_DS109\WObj:=Workobject_2;
  ENDPROC
  PROC Path_220()
    MoveL Target_3740_line3_starts,v1000,z100,ToolM_DS109\WObj:=Workobject_2;
    MoveL Target_3750,v1000,z100,ToolM_DS109\WObj:=Workobject_2;
    MoveL Target_3760,v1000,z100,ToolM_DS109\WObj:=Workobject_2;
    MoveL Target_3770,v1000,z100,ToolM_DS109\WObj:=Workobject_2;
    MoveL Target_3780,v1000,z100,ToolM_DS109\WObj:=Workobject_2;
    MoveL Target_3790,v1000,z100,ToolM_DS109\WObj:=Workobject_2;
    MoveL Target_3800,v1000,z100,ToolM_DS109\WObj:=Workobject_2;
    MoveL Target_3810,v1000,z100,ToolM_DS109\WObj:=Workobject_2;
    MoveL Target_3820,v1000,z100,ToolM_DS109\WObj:=Workobject_2;
    MoveL Target_3830,v1000,z100,ToolM_DS109\WObj:=Workobject_2;
    MoveL Target_3840,v1000,z100,ToolM_DS109\WObj:=Workobject_2;
    MoveL Target_3850,v1000,z100,ToolM_DS109\WObj:=Workobject_2;
    MoveL Target_3860,v1000,z100,ToolM_DS109\WObj:=Workobject_2;
    MoveL Target_3870,v1000,z100,ToolM_DS109\WObj:=Workobject_2;
    MoveL Target_3880_line3_ends,v1000,z100,ToolM_DS109\WObj:=Workobject_2;
  ENDPROC
ENDMODULE

